DATA_BLOCK "DB3326"
TITLE ==CH2++ZNE05_Alarm_List
{ S7_language := '16(1) Italiano (Italia)  10.08.2015  13:02:09' }
VERSION : 0.1


  STRUCT
   CM_ID : STRING  [8 ] := '=CH2_4';	//IDENTIFICATIVO TRATTO
   STATION_ID : STRING  [8 ] := '++ZNE05';	//TRATTO - ZONA - STAZIONE
   ELEMENT_ID : STRING  [8 ];	//ELEMENTO
   DB_ID : INT  := 3;	//GRANDEZZA DB O TIPO
   PART_IDENTIFICATION : STRING  [12 ];	//IDENTIFICAZIONE PEZZO IN LAVORAZIONE
   ACT_CYCLE_TIME : INT ;	//TEMPO CICLO EFFETTIVO
   COUNT_GOOD : INT ;	//PEZZO PRODOTTO BUONO
   COUNT_SCRAP : INT ;	//PEZZO PRODOTTO DI SCARTO
   ACCUMULATORS : ARRAY  [0 .. 15 ] OF //ACCUMULI
   INT ;
   SPARE_01 : ARRAY  [0 .. 17 ] OF //RISERVE
   INT ;
   CODE_EVENT : ARRAY  [0 .. 7 ] OF //CODICI DI DIAGNOSTICA (codici a 4 cifre)
   INT ;
   EVENTS : STRUCT 	//EVENTI DI DIAGNOSTICA / MONITORAGGIO (bit)
    E0001 : BOOL ;	//=CH2_4++ZNE05+HCZ01-DMC01;FALHA NO MÓDULO ET200S;1
    E0002 : BOOL ;	//=CH2_4++ZNE05+HCZ01-DSW01;FALHA DE SCALANCE;1
    E0003 : BOOL ;	//=CH2_4++ZNE05+HCZ01-QF_06;ALIMENTAÇÃO DISJUNTOR TÉRMICO PARA CIRCUITOS AUXILIARES;1
    E0004 : BOOL ;	//=CH2_4++ZNE05+HCZ01-QF_07;DISJUNTOR TÉRMICO. PODER COMANDOS E SINAIS DE SAÍDA;1
    E0005 : BOOL ;	//=CH2_4++ZNE05+HCZ01-QF_08;FONTE DE ALIMENTAÇÃO MAGNETOTÉRMICA PARA CIRCUITOS DE SEGURANÇA;1
    E0006 : BOOL ;	//=CH2_4++ZNE05+HCZ01-QF_09;DISJUNTOR TÉRMICO. PODER MÓDULOS E SWITCHES E/S ET200;1
    E0007 : BOOL ;
    E0008 : BOOL ;
    E0009 : BOOL ;
    E0010 : BOOL ;
    E0011 : BOOL ;
    E0012 : BOOL ;
    E0013 : BOOL ;
    E0014 : BOOL ;
    E0015 : BOOL ;
    E0016 : BOOL ;
    E0017 : BOOL ;	//=CH2_4++ZNE05+HCZ01-QF_10;FONTE DE ALIMENTAÇÃO 24VDC MOVIFIT FC01-FC02-FC03-FC04;1
    E0018 : BOOL ;	//=CH2_4++ZNE05+HCZ01-QF_11;24Vdc MOVIFIT FC05-06-07-08-09-10 SEP_04;1
    E0019 : BOOL ;	//=CH2_4++ZNE05+HCZ01-QF_20;440Vac MOVIFIT FC01 SETOR MOTOR 1 ZONA 5;1
    E0020 : BOOL ;	//=CH2_4++ZNE05+HCZ01-QF_21;440Vac MOVIFIT FC02 MOTOR SETOR 1 ZONA 5;1
    E0021 : BOOL ;	//=CH2_4++ZNE05+HCZ01-QF_22;FONTE DE ALIMENTAÇÃO 440Vac PARA MOTOR DA PLATAFORMA ESB01 SETOR 1;1
    E0022 : BOOL ;	//=CH2_4++ZNE05+HCZ01-QF_23;440Vac MOVIFIT FC03 MOTOR SETOR 2 ZONA 5;1
    E0023 : BOOL ;	//=CH2_4++ZNE05+HCZ01-QF_24;440Vac MOVIFIT FC04 MOTOR SETOR 3 ZONA 5;1
    E0024 : BOOL ;	//=CH2_4++ZNE05+HCZ01-QF_25;440Vca MOT. MOVIFIT FC05 - 06 - 07 SET. 4 ZONA 5;1
    E0025 : BOOL ;	//=CH2_4++ZNE05+HCZ01-QF_26;FONTE DE ALIMENTAÇÃO 440Vac PARA MOTOR PLATAFORMA ESB02, SETOR 4;1
    E0026 : BOOL ;	//=CH2_4++ZNE05+HCZ01-QF_27;440Vca MOT. MOVIFIT FC08 - 09 - 10 SEMANAS 5 ZONA 5;1
    E0027 : BOOL ;	//=CH2_4++ZNE05+HCZ01-KMS02;MOVIFIT FC01 SETOR DE EFICIÊNCIA DO RELÉ 1;1
    E0028 : BOOL ;	//=CH2_4++ZNE05+HCZ01-KMS04;EFICIÊNCIA DO RELÉ FC02 +ESB01 SETOR 1;1
    E0029 : BOOL ;	//=CH2_4++ZNE05+HCZ01-KMS06;MOVIFIT FC03 SETOR DE EFICIÊNCIA DO RELÉ 2;1
    E0030 : BOOL ;	//=CH2_4++ZNE05+HCZ01-KMS08;MOVIFIT FC04 SETOR DE EFICIÊNCIA DO RELÉ 3;1
    E0031 : BOOL ;	//=CH2_4++ZNE05+HCZ01-KMS010;EFICIÊNCIA DO RELÉ FC05 - 06 - 07 SETOR 4;1
    E0032 : BOOL ;	//=CH2_4++ZNE05+HCZ01-KMS012;EFICIÊNCIA DO RELÉ FC08 - 09 - 10 SETOR 5;1
    E0033 : BOOL ;	//=CH2_4++ZNE05+PTZ01-DMC01;FALHA NO MÓDULO ET200S;1
    E0034 : BOOL ;	//=CH2_4++ZNE05+PTZ02-DMC01;FALHA NO MÓDULO ET200S;1
    E0035 : BOOL ;	//=CH2_4++ZNE05+HKL01-DMC01;FALHA NO MÓDULO ET200S;1
    E0036 : BOOL ;	//=CH2_4++ZNE05+HKL02-DMC01;FALHA NO MÓDULO ET200S;1
    E0037 : BOOL ;	//=CH2_4++ZNE05+PLS01;FALHA DO SCANNER LASER;1
    E0038 : BOOL ;	//=CH2_4++ZNE05+PLS02;FALHA DO SCANNER LASER;1
    E0039 : BOOL ;	//=CH2_4++ZNE05+PLS03;FALHA DO SCANNER LASER;1
    E0040 : BOOL ;	//=CH2_4++ZNE05+PLS04;FALHA DO SCANNER LASER;1
    E0041 : BOOL ;	//=CH2_4++ZNE05+HCZ01-QF_28;FONTE DE ALIMENTAÇÃO 440Vac PARA MOTOR DA PLATAFORMA ESB03 SETOR 1;1
    E0042 : BOOL ;	//=CH2_4++ZNE05+HCZ01-KMS014;ESB03 SETOR DE EFICIÊNCIA DE RELÉ 1;1
    E0043 : BOOL ;	//=CH2_4++ZNE05+XGA01-SC_01;PORTÃO EM ANOMALIA;1
    E0044 : BOOL ;
    E0045 : BOOL ;
    E0046 : BOOL ;
    E0047 : BOOL ;
    E0048 : BOOL ;
    E0049 : BOOL ;
    E0050 : BOOL ;
    E0051 : BOOL ;
    E0052 : BOOL ;
    E0053 : BOOL ;
    E0054 : BOOL ;
    E0055 : BOOL ;
    E0056 : BOOL ;
    E0057 : BOOL ;
    E0058 : BOOL ;
    E0059 : BOOL ;
    E0060 : BOOL ;
    E0061 : BOOL ;
    E0062 : BOOL ;
    E0063 : BOOL ;
    E0064 : BOOL ;
    E0065 : BOOL ;
    E0066 : BOOL ;
    E0067 : BOOL ;
    E0068 : BOOL ;
    E0069 : BOOL ;
    E0070 : BOOL ;
    E0071 : BOOL ;
    E0072 : BOOL ;
    E0073 : BOOL ;
    E0074 : BOOL ;
    E0075 : BOOL ;
    E0076 : BOOL ;
    E0077 : BOOL ;
    E0078 : BOOL ;
    E0079 : BOOL ;
    E0080 : BOOL ;
    E0081 : BOOL ;	//=CH2_4++ZNE05+PTZ01-SB_07;BOTÃO DE EMERGENCIA APERTADO;2
    E0082 : BOOL ;	//=CH2_4++ZNE05+PTZ01-SB_07;EMERGÊNCIA NÃO RESTAURADA;2
    E0083 : BOOL ;	//=CH2_4++ZNE05+PTZ02-SB_07;BOTÃO DE EMERGENCIA APERTADO;2
    E0084 : BOOL ;	//=CH2_4++ZNE05+PTZ02-SB_07;EMERGÊNCIA NÃO RESTAURADA;2
    E0085 : BOOL ;	//=CH2_4++ZNE05+XGA01-SC_01;ACESSO ABERTO NÃO PROGRAMADO (GM);2
    E0086 : BOOL ;	//=CH2_4++ZNE05+XGA01-SC_01;ACESSO NÃO RESTAURADO(GM);2
    E0087 : BOOL ;	//=CH2_4++ZNE05+PRB03-BR_01;BARREIRA INTERDITADA;2
    E0088 : BOOL ;	//=CH2_4++ZNE05+PRB03-BR_01;BARREIRA NÃO RESTAURADA;2
    E0089 : BOOL ;	//=CH2_4++ZNE05+PRB04-BR_02;BARREIRA INTERDITADA;2
    E0090 : BOOL ;	//=CH2_4++ZNE05+PRB04-BR_02;BARREIRA NÃO RESTAURADA;2
    E0091 : BOOL ;	//=CH2_4++ZNE05+PRB01-BR_03;BARREIRA INTERDITADA;2
    E0092 : BOOL ;	//=CH2_4++ZNE05+PRB01-BR_03;BARREIRA NÃO RESTAURADA;2
    E0093 : BOOL ;	//=CH2_4++ZNE05+PRB02-VT_02;BARREIRA INTERDITADA;2
    E0094 : BOOL ;	//=CH2_4++ZNE05+PRB02-VT_02;BARREIRA NÃO RESTAURADA;2
    E0095 : BOOL ;	//=CH2_4++ZNE05+PLS01;SCANNER LASER OCUPADO;2
    E0096 : BOOL ;	//=CH2_4++ZNE05+PLS01;SCANNER LASER NÃO RESTAURADO;2
    E0097 : BOOL ;	//=CH2_4++ZNE05+PLS02;SCANNER LASER OCUPADO;2
    E0098 : BOOL ;	//=CH2_4++ZNE05+PLS02;SCANNER LASER NÃO RESTAURADO;2
    E0099 : BOOL ;	//=CH2_4++ZNE05+PLS03;SCANNER LASER OCUPADO;2
    E0100 : BOOL ;	//=CH2_4++ZNE05+PLS03;SCANNER LASER NÃO RESTAURADO;2
    E0101 : BOOL ;	//=CH2_4++ZNE05+PLS04;SCANNER LASER OCUPADO;2
    E0102 : BOOL ;	//=CH2_4++ZNE05+PLS04;SCANNER LASER NÃO RESTAURADO;2
    E0103 : BOOL ;	//=CH2_4++ZNE05+SLL01-SB_01;BOTÃO DE EMERGENCIA APERTADO;2
    E0104 : BOOL ;	//=CH2_4++ZNE05+SLL01-SB_01;EMERGÊNCIA NÃO RESTAURADA;2
    E0105 : BOOL ;	//=CH2_4++ZNE05+SLL02-SB_01;BOTÃO DE EMERGENCIA APERTADO;2
    E0106 : BOOL ;	//=CH2_4++ZNE05+SLL02-SB_01;EMERGÊNCIA NÃO RESTAURADA;2
    E0107 : BOOL ;	//=CH2_4++ZNE05+PEM01-SB_01;BOTÃO DE EMERGENCIA APERTADO;2
    E0108 : BOOL ;	//=CH2_4++ZNE05+PEM01-SB_01;EMERGÊNCIA NÃO RESTAURADA;2
    E0109 : BOOL ;	//=CH2_4++ZNE05+PEM02-SB_01;BOTÃO DE EMERGENCIA APERTADO;2
    E0110 : BOOL ;	//=CH2_4++ZNE05+PEM02-SB_01;EMERGÊNCIA NÃO RESTAURADA;2
    E0111 : BOOL ;	//=CH2_4++ZNE05+PSC01-SB_01;BOTÃO DE EMERGENCIA APERTADO;2
    E0112 : BOOL ;	//=CH2_4++ZNE05+PSC01-SB_01;EMERGÊNCIA NÃO RESTAURADA;2
    E0113 : BOOL ;	//=CH2_4++ZNE05+PSC02-SB_01;BOTÃO DE EMERGENCIA APERTADO;2
    E0114 : BOOL ;	//=CH2_4++ZNE05+PSC02-SB_01;EMERGÊNCIA NÃO RESTAURADA;2
    E0115 : BOOL ;	//=CH2_4++ZNE05+PSC03-SB_01;BOTÃO DE EMERGENCIA APERTADO;2
    E0116 : BOOL ;	//=CH2_4++ZNE05+PSC03-SB_01;EMERGÊNCIA NÃO RESTAURADA;2
    E0117 : BOOL ;
    E0118 : BOOL ;
    E0119 : BOOL ;	//=CH2_4++ZNE05+XGA01-SC_01;MANUTENÇÃO PROGRAMADA DE ACESSO ABERTO (PM);13
    E0120 : BOOL ;	//=CH2_4++ZNE05+XGA01-SC_01;LIMPEZA TÉCNICA DE ACESSO ABERTO (AM);14
    E0121 : BOOL ;	//=CH2_4++ZNE05+XGA01-SC_01;ACESSO NÃO RESTAURADO PROG. DE MANUTENÇÃO (PM);13
    E0122 : BOOL ;	//=CH2_4++ZNE05+XGA01-SC_01;ACESSO NÃO RESTAURADO LIMPEZA TÉCNICA (AM);14
    E0123 : BOOL ;	//=CH2_4++ZNE05+OIB01-SB_01;BOTÃO DE EMERGENCIA APERTADO;2
    E0124 : BOOL ;	//=CH2_4++ZNE05+OIB01-SB_01;EMERGÊNCIA NÃO RESTAURADA;2
    E0125 : BOOL ;
    E0126 : BOOL ;
    E0127 : BOOL ;
    E0128 : BOOL ;
    E0129 : BOOL ;	//=CH2_4++ZNE05+HCZ01-QF_03;FONTE DE ALIMENTAÇÃO MAGNETOTÉRMICA PARA AR CONDICIONADO 400V;58
    E0130 : BOOL ;	//=CH2_4++ZNE05+HCZ01-QF_15;MAGNETO. PODER PAINEL OPERADOR 24Vdc +PTZ01;58
    E0131 : BOOL ;	//=CH2_4++ZNE05+HCZ01-QF_16;MAGNETO. PODER PAINEL OPERADOR 24Vdc +PTZ02;58
    E0132 : BOOL ;	//=CH2_4++ZNE05+PTZ01-DSP01;PRÉ-ALARME SEM PLC <-> COMUNICAÇÃO IHM;58
    E0133 : BOOL ;	//=CH2_4++ZNE05+PTZ02-DSP01;PRÉ-ALARME SEM PLC <-> COMUNICAÇÃO IHM;58
    E0134 : BOOL ;	//=CH2_4++ZNE05+PTZ01-SA_03;PEDIDO DE ACESSO PARA MANUTENÇÃO PLANEJADA (PM);58
    E0135 : BOOL ;	//=CH2_4++ZNE05+PTZ01-SA_03;SOLICITAR ACESSO PARA LIMPEZA TÉCNICA (AM);58
    E0136 : BOOL ;	//=CH2_4++ZNE05+PTZ02-SA_03;PEDIDO DE ACESSO PARA MANUTENÇÃO PLANEJADA (PM);58
    E0137 : BOOL ;	//=CH2_4++ZNE05+PTZ02-SA_03;SOLICITAR ACESSO PARA LIMPEZA TÉCNICA (AM);58
    E0138 : BOOL ;	//=CH2_4++ZNE05+PTZ01-SA_03;SOLICITAR ACESSO PARA MANUTENÇÃO NÃO PROGRAMADA (GM);58
    E0139 : BOOL ;	//=CH2_4++ZNE05+PTZ02-SA_03;SOLICITAR ACESSO PARA MANUTENÇÃO NÃO PROGRAMADA (GM);58
    E0140 : BOOL ;	//=CH2_4++ZNE05+HCZ01-ST_01;CONTROLE DE TEMPERATURA DO GABINETE;58
    E0141 : BOOL ;	//=CH2_4++ZNE05+PLS01;SCANNER LASER EM PRÉ-ALARME;58
    E0142 : BOOL ;	//=CH2_4++ZNE05+PLS02;SCANNER LASER EM PRÉ-ALARME;58
    E0143 : BOOL ;	//=CH2_4++ZNE05+PLS03;SCANNER LASER EM PRÉ-ALARME;58
    E0144 : BOOL ;	//=CH2_4++ZNE05+PLS04;SCANNER LASER EM PRÉ-ALARME;58
    E0145 : BOOL ;	//=CH2_4++ZNE05+PTZ01;SETOR ASCENTE NÃO ESTÁ EM CICLO INICIADO;58
    E0146 : BOOL ;	//=CH2_4++ZNE05+PTZ01;SETOR JUSANTE NÃO ESTÁ EM CICLO INICIADO;58
    E0147 : BOOL ;	//=CH2_4++ZNE05+PTZ02;SETOR ASCENTE NÃO ESTÁ EM CICLO INICIADO;58
    E0148 : BOOL ;	//=CH2_4++ZNE05+PTZ02;SETOR JUSANTE NÃO ESTÁ EM CICLO INICIADO;58
    E0149 : BOOL ;	//=CH2_4++ZNE05+PTZ03;SETOR ASCENTE NÃO ESTÁ EM CICLO INICIADO;58
    E0150 : BOOL ;	//=CH2_4++ZNE05+PTZ03;SETOR JUSANTE NÃO ESTÁ EM CICLO INICIADO;58
    E0151 : BOOL ;	//=CH2_4++ZNE05+PRE01;SETOR ASCENTE NÃO ESTÁ EM CICLO INICIADO;58
    E0152 : BOOL ;	//=CH2_4++ZNE05+PRE01;SETOR JUSANTE NÃO ESTÁ EM CICLO INICIADO;58
    E0153 : BOOL ;	//=CH2_4++ZNE05+HCZ01;PRÉ-ALARME DE SEGURANÇA DE BYPASS ATIVO;54
    E0154 : BOOL ;	//=CH2_4++ZNE05+TTS06;NKE WARNING TROCA CARTA DE LIMPEZA;4
    E0155 : BOOL ;	//=CH2_4++ZNE05+TTS06;ALARME TROCA DO CARTÃO NKE LIMPEZA;3
    E0156 : BOOL ;	//=CH2_4++ZNE05+LM07;PARCEIRO DE BATERIA DO FIM DE CURSO ACIONADO;10
    E0157 : BOOL ;
    E0158 : BOOL ;
    E0159 : BOOL ;
    E0160 : BOOL ;
    E0161 : BOOL ;
    E0162 : BOOL ;
    E0163 : BOOL ;
    E0164 : BOOL ;
    E0165 : BOOL ;
    E0166 : BOOL ;
    E0167 : BOOL ;
    E0168 : BOOL ;
    E0169 : BOOL ;
    E0170 : BOOL ;
    E0171 : BOOL ;
    E0172 : BOOL ;
    E0173 : BOOL ;
    E0174 : BOOL ;
    E0175 : BOOL ;
    E0176 : BOOL ;
    E0177 : BOOL ;	//=CH2_4++ZNE05+OIB01-DMC01;ANOMALIA DO MÓDULO ProfSafe ET200S-FDI-FDO;2
    E0178 : BOOL ;	//=CH2_4++ZNE05+HCZ01-DMC01;ANOMALIA DO MÓDULO ProfSafe ET200S-FDI-FDO;2
    E0179 : BOOL ;	//=CH2_4++ZNE05+PTZ01-DMC01;ANOMALIA DO MÓDULO ProfSafe ET200S-FDI;2
    E0180 : BOOL ;	//=CH2_4++ZNE05+PTZ02-DMC01;ANOMALIA DO MÓDULO ProfSafe ET200S-FDI;2
    E0181 : BOOL ;	//=CH2_4++ZNE05+PTZ03-DMC01;ANOMALIA DO MÓDULO ProfSafe ET200S-FDI;2
    E0182 : BOOL ;	//=CH2_4++ZNE05+PRE01-DMC01;ANOMALIA DO MÓDULO ProfSafe ET200S-FDI;2
    E0183 : BOOL ;	//=CH2_4++ZNE05+HKL01-DMC01;ANOMALIA DO MÓDULO ProfSafe ET200S-FDI;2
    E0184 : BOOL ;	//=CH2_4++ZNE05+HKL02-DMC01;ANOMALIA DO MÓDULO ProfSafe ET200S-FDI;2
    E0185 : BOOL ;	//=CH2_4++ZNE05+HCZ02-DMC01;ANOMALIA DO MÓDULO ProfSafe ET200S-FDI-FDO;2
    E0186 : BOOL ;
    E0187 : BOOL ;
    E0188 : BOOL ;
    E0189 : BOOL ;
    E0190 : BOOL ;
    E0191 : BOOL ;
    E0192 : BOOL ;
    E0193 : BOOL ;
    E0194 : BOOL ;
    E0195 : BOOL ;
    E0196 : BOOL ;
    E0197 : BOOL ;
    E0198 : BOOL ;
    E0199 : BOOL ;
    E0200 : BOOL ;
    E0201 : BOOL ;
    E0202 : BOOL ;
    E0203 : BOOL ;
    E0204 : BOOL ;
    E0205 : BOOL ;
    E0206 : BOOL ;
    E0207 : BOOL ;
    E0208 : BOOL ;
    E0209 : BOOL ;	//=CH2_4++ZNE05;EM PRODUÇÃO;19
    E0210 : BOOL ;	//=CH2_4++ZNE05+PTZ01-SB_05;INICIAR CICLO AUTOMÁTICO;15
    E0211 : BOOL ;	//=CH2_4++ZNE05+PTZ02-SB_05;INICIAR CICLO AUTOMÁTICO;15
    E0212 : BOOL ;	//=CH2_4++ZNE05+PTZ01-SA_01;CICLO MANUAL SELECIONADO;16
    E0213 : BOOL ;	//=CH2_4++ZNE05+PTZ02-SA_01;CICLO MANUAL SELECIONADO;16
    E0214 : BOOL ;	//=CH2_4++ZNE05+PTZ01-SB_04;PARADA DO CICLO;17
    E0215 : BOOL ;	//=CH2_4++ZNE05+PTZ02-SB_04;PARADA DO CICLO;17
    E0216 : BOOL ;
    E0217 : BOOL ;	//=CH2_4++ZNE05+TTS01;FALHA NO CARREGAMENTO;6
    E0218 : BOOL ;	//=CH2_4++ZNE05+TTS12;FALHA NO DESCARREGAMENTO;9
    E0219 : BOOL ;	//=CH2_4++ZNE05+TTS04;OPERADOR DE SOBRECICLO;8
    E0220 : BOOL ;	//=CH2_4++ZNE05+TTS05;OPERADOR DE SOBRECICLO;8
    E0221 : BOOL ;
    E0222 : BOOL ;
    E0223 : BOOL ;
    E0224 : BOOL ;
    E0225 : BOOL ;	//=CH2_4++ZNE05+TTS01-SQA01;FALHA NO INTERRUPTOR DE LIMITE DE PARADA;1
    E0226 : BOOL ;	//=CH2_4++ZNE05+TTS01-SQS01;FALHA NO INTERRUPTOR DE LIMITE DE LENTAÇÃO;1
    E0227 : BOOL ;	//=CH2_4++ZNE05+TTS01-SQC01;FALHA NO INTERRUPTOR DE LIMITE DE CONTROLE DE POSIÇÃO;1
    E0228 : BOOL ;	//=CH2_4++ZNE05+TTS01-B__01;FALHA DA FOTOCÉLULA NA PRESENÇA DO VEÍCULO;1
    E0229 : BOOL ;	//=CH2_4++ZNE05+TTS01;SAIR DO TEMPO DE TRANSFERÊNCIA;1
    E0230 : BOOL ;	//=CH2_4++ZNE05+TTS01;CTRL ENGRENAGEM TTS ANTERIOR;1
    E0231 : BOOL ;	//=CH2_4++ZNE05+TTS01;CTRL ENGRENAGEM PRÓXIMO TTS;1
    E0232 : BOOL ;	//=CH2_4++ZNE05+TTS01;POSIÇÃO CTRL;1
    E0233 : BOOL ;	//=CH2_4++ZNE05+TTS01-M__01;FALHA NO INVERSOR;1
    E0234 : BOOL ;	//=CH2_4++ZNE05+TTS01-M__01;ERRO DE COMUNICAÇÃO DO INVERSOR;1
    E0235 : BOOL ;	//=CH2_4++ZNE05+TTS01-SQA02;FALHA DO INTERRUPTOR DE LIMITE DE PROTEÇÃO QUEDA TRABALHO FECHADO;1
    E0236 : BOOL ;	//=CH2_4++ZNE05+TTS01-SQB02;FALHA DE RESTO ABERTO DO INTERRUPTOR DE LIMITE DE PROTEÇÃO QUEDA;1
    E0237 : BOOL ;	//=CH2_4++ZNE05+TTS01-SQ_01;QUEBRA DA CORREIA DE TRANSMISSÃO TTS;1
    E0238 : BOOL ;	//=CH2_4++ZNE05+TTS01;PRÉ-ALARME DE BYPASS DE FALHA ATIVO;58
    E0239 : BOOL ;	//=CH2_4++ZNE05+TTS01-M__01;PRÉ-ALARME DE CORRENTE ABSORVIDA;58
    E0240 : BOOL ;	//=CH2_4++ZNE05+TTS01-M__01;PRÉ-ALARME DO INVERSOR MOVIMOT;58
    E0241 : BOOL ;	//=CH2_4++ZNE05+TTS01-U__01;ERRO DE COMUNICAÇÃO MOVIFIT;1
    E0242 : BOOL ;	//=CH2_4++ZNE05+TTS01-U__01;INTERRUPTOR MOVIFIT ABERTO 380V;1
    E0243 : BOOL ;	//=CH2_4++ZNE05+TTS01-U__01;AUSÊNCIAS 24 VOLTS MOVIFIT SEGURANÇA;1
    E0244 : BOOL ;	//=CH2_4++ZNE05+TTS01-U__01;AUSÊNCIAS MOVIFIT 24 VOLT;1
    E0245 : BOOL ;	//=CH2_4++ZNE05+TTS01-U__01;ANOMALIA MOVIFIT;1
    E0246 : BOOL ;	//=CH2_4++ZNE05+TTS01-U__01;SOBRECARGA DE TENSÃO DE SAÍDA 0 MOVIFIT;1
    E0247 : BOOL ;	//=CH2_4++ZNE05+TTS01-U__01;TENSÃO DE SAÍDA DE SOBRECARGA SAÍDA 1 MOVIFIT;1
    E0248 : BOOL ;	//=CH2_4++ZNE05+TTS01-U__01;SOBRECARGA DE TENSÃO DO MOVIFIT NA SAÍDA 2;1
    E0249 : BOOL ;	//=CH2_4++ZNE05+TTS01-U__01;SOBRECARGA DE TENSÃO DE SAÍDA 3 MOVIFIT;1
    E0250 : BOOL ;	//=CH2_4++ZNE05+TTS01-U__01;SOBRECARGA DE TENSÃO DO SENSOR MOVIFIT GRUPO 1;1
    E0251 : BOOL ;	//=CH2_4++ZNE05+TTS01-U__01;SOBRECARGA DE TENSÃO DO SENSOR MOVIFIT GRUPO 2;1
    E0252 : BOOL ;	//=CH2_4++ZNE05+TTS01-U__01;SOBRECARGA DE TENSÃO DO SENSOR MOVIFIT GRUPO 3;1
    E0253 : BOOL ;	//=CH2_4++ZNE05+TTS01-U__01;SOBRECARGA DE TENSÃO DO SENSOR MOVIFIT GRUPO 4;1
    E0254 : BOOL ;
    E0255 : BOOL ;
    E0256 : BOOL ;
    E0257 : BOOL ;	//=CH2_4++ZNE05+TTS02-SQA01;FALHA NO INTERRUPTOR DE LIMITE DE PARADA;1
    E0258 : BOOL ;	//=CH2_4++ZNE05+TTS02-SQS01;FALHA NO INTERRUPTOR DE LIMITE DE LENTAÇÃO;1
    E0259 : BOOL ;	//=CH2_4++ZNE05+TTS02-SQC01;FALHA NO INTERRUPTOR DE LIMITE DE CONTROLE DE POSIÇÃO;1
    E0260 : BOOL ;	//=CH2_4++ZNE05+TTS02-B__01;FALHA DA FOTOCÉLULA NA PRESENÇA DO VEÍCULO;1
    E0261 : BOOL ;	//=CH2_4++ZNE05+TTS02;SAIR DO TEMPO DE TRANSFERÊNCIA;1
    E0262 : BOOL ;	//=CH2_4++ZNE05+TTS02;CTRL ENGRENAGEM TTS ANTERIOR;1
    E0263 : BOOL ;	//=CH2_4++ZNE05+TTS02;CTRL ENGRENAGEM PRÓXIMO TTS;1
    E0264 : BOOL ;	//=CH2_4++ZNE05+TTS02;POSIÇÃO CTRL;1
    E0265 : BOOL ;	//=CH2_4++ZNE05+TTS02-M__01;FALHA NO INVERSOR;1
    E0266 : BOOL ;	//=CH2_4++ZNE05+TTS02-M__01;ERRO DE COMUNICAÇÃO DO INVERSOR;1
    E0267 : BOOL ;	//=CH2_4++ZNE05+TTS02-SQA02;FALHA DO INTERRUPTOR DE LIMITE DE PROTEÇÃO QUEDA TRABALHO FECHADO;1
    E0268 : BOOL ;	//=CH2_4++ZNE05+TTS02-SQB02;FALHA DE RESTO ABERTO DO INTERRUPTOR DE LIMITE DE PROTEÇÃO QUEDA;1
    E0269 : BOOL ;	//=CH2_4++ZNE05+TTS02-SQ_01;QUEBRA DA CORREIA DE TRANSMISSÃO TTS;1
    E0270 : BOOL ;	//=CH2_4++ZNE05+TTS02;PRÉ-ALARME DE BYPASS DE FALHA ATIVO;58
    E0271 : BOOL ;	//=CH2_4++ZNE05+TTS02-M__01;PRÉ-ALARME DE CORRENTE ABSORVIDA;58
    E0272 : BOOL ;	//=CH2_4++ZNE05+TTS02-M__01;PRÉ-ALARME DO INVERSOR MOVIMOT;58
    E0273 : BOOL ;	//=CH2_4++ZNE05+TTS02-U__01;ERRO DE COMUNICAÇÃO MOVIFIT;1
    E0274 : BOOL ;	//=CH2_4++ZNE05+TTS02-U__01;INTERRUPTOR MOVIFIT ABERTO 380V;1
    E0275 : BOOL ;	//=CH2_4++ZNE05+TTS02-U__01;AUSÊNCIAS 24 VOLTS MOVIFIT SEGURANÇA;1
    E0276 : BOOL ;	//=CH2_4++ZNE05+TTS02-U__01;AUSÊNCIAS MOVIFIT 24 VOLT;1
    E0277 : BOOL ;	//=CH2_4++ZNE05+TTS02-U__01;ANOMALIA MOVIFIT;1
    E0278 : BOOL ;	//=CH2_4++ZNE05+TTS02-U__01;SOBRECARGA DE TENSÃO DE SAÍDA 0 MOVIFIT;1
    E0279 : BOOL ;	//=CH2_4++ZNE05+TTS02-U__01;TENSÃO DE SAÍDA DE SOBRECARGA SAÍDA 1 MOVIFIT;1
    E0280 : BOOL ;	//=CH2_4++ZNE05+TTS02-U__01;SOBRECARGA DE TENSÃO DO MOVIFIT NA SAÍDA 2;1
    E0281 : BOOL ;	//=CH2_4++ZNE05+TTS02-U__01;SOBRECARGA DE TENSÃO DE SAÍDA 3 MOVIFIT;1
    E0282 : BOOL ;	//=CH2_4++ZNE05+TTS02-U__01;SOBRECARGA DE TENSÃO DO SENSOR MOVIFIT GRUPO 1;1
    E0283 : BOOL ;	//=CH2_4++ZNE05+TTS02-U__01;SOBRECARGA DE TENSÃO DO SENSOR MOVIFIT GRUPO 2;1
    E0284 : BOOL ;	//=CH2_4++ZNE05+TTS02-U__01;SOBRECARGA DE TENSÃO DO SENSOR MOVIFIT GRUPO 3;1
    E0285 : BOOL ;	//=CH2_4++ZNE05+TTS02-U__01;SOBRECARGA DE TENSÃO DO SENSOR MOVIFIT GRUPO 4;1
    E0286 : BOOL ;
    E0287 : BOOL ;
    E0288 : BOOL ;
    E0289 : BOOL ;	//=CH2_4++ZNE05+ESB01-SQA01;FALHA NO INTERRUPTOR DE LIMITE DE PARAGEM INFERIOR DA PLATAFORMA MÓVEL +ESB;1
    E0290 : BOOL ;	//=CH2_4++ZNE05+ESB01-SQB01;FALHA NO INTERRUPTOR DE LIMITE DE PARADA ALTA DA PLATAFORMA MÓVEL +ESB;1
    E0291 : BOOL ;
    E0292 : BOOL ;
    E0293 : BOOL ;	//=CH2_4++ZNE05+ESB01-SQA01;TIME OUT DESCIDA +ESB;1
    E0294 : BOOL ;	//=CH2_4++ZNE05+ESB01-SQB01;TIME OUT RISE +ESB;1
    E0295 : BOOL ;
    E0296 : BOOL ;
    E0297 : BOOL ;	//=CH2_4++ZNE05+ESB01-HKM03;SONDA TÉRMICA DO MOTOR +ESB;1
    E0298 : BOOL ;
    E0299 : BOOL ;
    E0300 : BOOL ;
    E0301 : BOOL ;
    E0302 : BOOL ;
    E0303 : BOOL ;
    E0304 : BOOL ;
    E0305 : BOOL ;	//=CH2_4++ZNE05+ESB01;ESTAÇÃO EXCLUÍDA PRÉ-ALARME;58
    E0306 : BOOL ;
    E0307 : BOOL ;
    E0308 : BOOL ;
    E0309 : BOOL ;
    E0310 : BOOL ;
    E0311 : BOOL ;
    E0312 : BOOL ;
    E0313 : BOOL ;	//=CH2_4++ZNE05+ESB01;PRÉ-ALARME DE BYPASS DE FALHA ATIVO;58
    E0314 : BOOL ;
    E0315 : BOOL ;
    E0316 : BOOL ;
    E0317 : BOOL ;
    E0318 : BOOL ;
    E0319 : BOOL ;
    E0320 : BOOL ;
    E0321 : BOOL ;	//=CH2_4++ZNE05+TTS03-SQA01;FALHA NO INTERRUPTOR DE LIMITE DE PARADA;1
    E0322 : BOOL ;	//=CH2_4++ZNE05+TTS03-SQS01;FALHA NO INTERRUPTOR DE LIMITE DE LENTAÇÃO;1
    E0323 : BOOL ;	//=CH2_4++ZNE05+TTS03-SQC01;FALHA NO INTERRUPTOR DE LIMITE DE CONTROLE DE POSIÇÃO;1
    E0324 : BOOL ;	//=CH2_4++ZNE05+TTS03-B__01;FALHA DA FOTOCÉLULA NA PRESENÇA DO VEÍCULO;1
    E0325 : BOOL ;	//=CH2_4++ZNE05+TTS03;SAIR DO TEMPO DE TRANSFERÊNCIA;1
    E0326 : BOOL ;	//=CH2_4++ZNE05+TTS03;CTRL ENGRENAGEM TTS ANTERIOR;1
    E0327 : BOOL ;	//=CH2_4++ZNE05+TTS03;CTRL ENGRENAGEM PRÓXIMO TTS;1
    E0328 : BOOL ;	//=CH2_4++ZNE05+TTS03;POSIÇÃO CTRL;1
    E0329 : BOOL ;	//=CH2_4++ZNE05+TTS03-M__01;FALHA NO INVERSOR;1
    E0330 : BOOL ;	//=CH2_4++ZNE05+TTS03-M__01;ERRO DE COMUNICAÇÃO DO INVERSOR;1
    E0331 : BOOL ;	//=CH2_4++ZNE05+TTS03-SQA02;FALHA DO INTERRUPTOR DE LIMITE DE PROTEÇÃO QUEDA TRABALHO FECHADO;1
    E0332 : BOOL ;	//=CH2_4++ZNE05+TTS03-SQB02;FALHA DE RESTO ABERTO DO INTERRUPTOR DE LIMITE DE PROTEÇÃO QUEDA;1
    E0333 : BOOL ;	//=CH2_4++ZNE05+TTS03-SQ_01;QUEBRA DA CORREIA DE TRANSMISSÃO TTS;1
    E0334 : BOOL ;	//=CH2_4++ZNE05+TTS03;PRÉ-ALARME DE BYPASS DE FALHA ATIVO;58
    E0335 : BOOL ;	//=CH2_4++ZNE05+TTS03-M__01;PRÉ-ALARME DE CORRENTE ABSORVIDA;58
    E0336 : BOOL ;	//=CH2_4++ZNE05+TTS03-M__01;PRÉ-ALARME DO INVERSOR MOVIMOT;58
    E0337 : BOOL ;	//=CH2_4++ZNE05+TTS03-U__01;ERRO DE COMUNICAÇÃO MOVIFIT;1
    E0338 : BOOL ;	//=CH2_4++ZNE05+TTS03-U__01;INTERRUPTOR MOVIFIT ABERTO 380V;1
    E0339 : BOOL ;	//=CH2_4++ZNE05+TTS03-U__01;AUSÊNCIAS 24 VOLTS MOVIFIT SEGURANÇA;1
    E0340 : BOOL ;	//=CH2_4++ZNE05+TTS03-U__01;AUSÊNCIAS MOVIFIT 24 VOLT;1
    E0341 : BOOL ;	//=CH2_4++ZNE05+TTS03-U__01;ANOMALIA MOVIFIT;1
    E0342 : BOOL ;	//=CH2_4++ZNE05+TTS03-U__01;SOBRECARGA DE TENSÃO DE SAÍDA 0 MOVIFIT;1
    E0343 : BOOL ;	//=CH2_4++ZNE05+TTS03-U__01;TENSÃO DE SAÍDA DE SOBRECARGA SAÍDA 1 MOVIFIT;1
    E0344 : BOOL ;	//=CH2_4++ZNE05+TTS03-U__01;SOBRECARGA DE TENSÃO DO MOVIFIT NA SAÍDA 2;1
    E0345 : BOOL ;	//=CH2_4++ZNE05+TTS03-U__01;SOBRECARGA DE TENSÃO DE SAÍDA 3 MOVIFIT;1
    E0346 : BOOL ;	//=CH2_4++ZNE05+TTS03-U__01;SOBRECARGA DE TENSÃO DO SENSOR MOVIFIT GRUPO 1;1
    E0347 : BOOL ;	//=CH2_4++ZNE05+TTS03-U__01;SOBRECARGA DE TENSÃO DO SENSOR MOVIFIT GRUPO 2;1
    E0348 : BOOL ;	//=CH2_4++ZNE05+TTS03-U__01;SOBRECARGA DE TENSÃO DO SENSOR MOVIFIT GRUPO 3;1
    E0349 : BOOL ;	//=CH2_4++ZNE05+TTS03-U__01;SOBRECARGA DE TENSÃO DO SENSOR MOVIFIT GRUPO 4;1
    E0350 : BOOL ;
    E0351 : BOOL ;
    E0352 : BOOL ;
    E0353 : BOOL ;	//=CH2_4++ZNE05+TTS04-SQA01;FALHA NO INTERRUPTOR DE LIMITE DE PARADA;1
    E0354 : BOOL ;	//=CH2_4++ZNE05+TTS04-SQS01;FALHA NO INTERRUPTOR DE LIMITE DE LENTAÇÃO;1
    E0355 : BOOL ;	//=CH2_4++ZNE05+TTS04-SQC01;FALHA NO INTERRUPTOR DE LIMITE DE CONTROLE DE POSIÇÃO;1
    E0356 : BOOL ;	//=CH2_4++ZNE05+TTS04-B__01;FALHA DA FOTOCÉLULA NA PRESENÇA DO VEÍCULO;1
    E0357 : BOOL ;	//=CH2_4++ZNE05+TTS04;SAIR DO TEMPO DE TRANSFERÊNCIA;1
    E0358 : BOOL ;	//=CH2_4++ZNE05+TTS04;CTRL ENGRENAGEM TTS ANTERIOR;1
    E0359 : BOOL ;	//=CH2_4++ZNE05+TTS04;CTRL ENGRENAGEM PRÓXIMO TTS;1
    E0360 : BOOL ;	//=CH2_4++ZNE05+TTS04;POSIÇÃO CTRL;1
    E0361 : BOOL ;	//=CH2_4++ZNE05+TTS04-M__01;FALHA NO INVERSOR;1
    E0362 : BOOL ;	//=CH2_4++ZNE05+TTS04-M__01;ERRO DE COMUNICAÇÃO DO INVERSOR;1
    E0363 : BOOL ;	//=CH2_4++ZNE05+TTS04-SQA02;FALHA DO INTERRUPTOR DE LIMITE DE PROTEÇÃO QUEDA TRABALHO FECHADO;1
    E0364 : BOOL ;	//=CH2_4++ZNE05+TTS04-SQB02;FALHA DE RESTO ABERTO DO INTERRUPTOR DE LIMITE DE PROTEÇÃO QUEDA;1
    E0365 : BOOL ;	//=CH2_4++ZNE05+TTS04-SQ_01;QUEBRA DA CORREIA DE TRANSMISSÃO TTS;1
    E0366 : BOOL ;	//=CH2_4++ZNE05+TTS04;PRÉ-ALARME DE BYPASS DE FALHA ATIVO;58
    E0367 : BOOL ;	//=CH2_4++ZNE05+TTS04-M__01;PRÉ-ALARME DE CORRENTE ABSORVIDA;58
    E0368 : BOOL ;	//=CH2_4++ZNE05+TTS04-M__01;PRÉ-ALARME DO INVERSOR MOVIMOT;58
    E0369 : BOOL ;	//=CH2_4++ZNE05+TTS04-U__01;ERRO DE COMUNICAÇÃO MOVIFIT;1
    E0370 : BOOL ;	//=CH2_4++ZNE05+TTS04-U__01;INTERRUPTOR MOVIFIT ABERTO 380V;1
    E0371 : BOOL ;	//=CH2_4++ZNE05+TTS04-U__01;AUSÊNCIAS 24 VOLTS MOVIFIT SEGURANÇA;1
    E0372 : BOOL ;	//=CH2_4++ZNE05+TTS04-U__01;AUSÊNCIAS MOVIFIT 24 VOLT;1
    E0373 : BOOL ;	//=CH2_4++ZNE05+TTS04-U__01;ANOMALIA MOVIFIT;1
    E0374 : BOOL ;	//=CH2_4++ZNE05+TTS04-U__01;SOBRECARGA DE TENSÃO DE SAÍDA 0 MOVIFIT;1
    E0375 : BOOL ;	//=CH2_4++ZNE05+TTS04-U__01;TENSÃO DE SAÍDA DE SOBRECARGA SAÍDA 1 MOVIFIT;1
    E0376 : BOOL ;	//=CH2_4++ZNE05+TTS04-U__01;SOBRECARGA DE TENSÃO DO MOVIFIT NA SAÍDA 2;1
    E0377 : BOOL ;	//=CH2_4++ZNE05+TTS04-U__01;SOBRECARGA DE TENSÃO DE SAÍDA 3 MOVIFIT;1
    E0378 : BOOL ;	//=CH2_4++ZNE05+TTS04-U__01;SOBRECARGA DE TENSÃO DO SENSOR MOVIFIT GRUPO 1;1
    E0379 : BOOL ;	//=CH2_4++ZNE05+TTS04-U__01;SOBRECARGA DE TENSÃO DO SENSOR MOVIFIT GRUPO 2;1
    E0380 : BOOL ;	//=CH2_4++ZNE05+TTS04-U__01;SOBRECARGA DE TENSÃO DO SENSOR MOVIFIT GRUPO 3;1
    E0381 : BOOL ;	//=CH2_4++ZNE05+TTS04-U__01;SOBRECARGA DE TENSÃO DO SENSOR MOVIFIT GRUPO 4;1
    E0382 : BOOL ;
    E0383 : BOOL ;
    E0384 : BOOL ;
    E0385 : BOOL ;	//=CH2_4++ZNE05+WIP01;PARADA DE LINHA DO MES/PLC PARA CHAMADA DE OPERADOR;11
    E0386 : BOOL ;	//=CH2_4++ZNE05+WIP01;NÓ PROFINET DO LEITOR NÃO ESTÁ OK;1
    E0387 : BOOL ;	//=CH2_4++ZNE05+WIP01;PLACA CODIFICADORA DE NÓ PROFINET NÃO OK;1
    E0388 : BOOL ;	//=CH2_4++ZNE05+WIP01;MAU FUNCIONAMENTO DO SENSOR DE PITCHING;1
    E0389 : BOOL ;	//=CH2_4++ZNE05+WIP01;DISFUNÇÃO DE TRÂNSITO DO PONTO DE AJUSTE;1
    E0390 : BOOL ;	//=CH2_4++ZNE05+WIP01;MAU FUNCIONAMENTO DO CODIFICADOR;1
    E0391 : BOOL ;
    E0392 : BOOL ;
    E0393 : BOOL ;	//=CH2_4++ZNE05+WIP01;ANOMALIA DE LEITURA DE CÓDIGO DE BARRAS/TAG;5
    E0394 : BOOL ;	//=CH2_4++ZNE05+WIP01;TEMPO ESGOTADO DE LEITURA DE CÓDIGO DE BARRAS/TAG;5
    E0395 : BOOL ;	//=CH2_4++ZNE05+WIP01;INCONSISTÊNCIA FÍSICO-LÓGICA;5
    E0396 : BOOL ;	//=CH2_4++ZNE05+WIP01;VERIFIQUE O DÍGITO ERRADO CIS;5
    E0397 : BOOL ;	//=CH2_4++ZNE05+WIP01;TEMPO LIMITE PARA RECEBIMENTO DE DADOS DO PERÍODO ANTERIOR;5
    E0398 : BOOL ;	//=CH2_4++ZNE05+WIP01;INCONSISTÊNCIA DE DADOS DE SET POINT CIS/VIS COM CIS/VIS NEXT;5
    E0399 : BOOL ;	//=CH2_4++ZNE05+WIP01;LINHA WIP DO SERVIÇO MES NÃO ATIVA (PARADA DE LINHA);10
    E0400 : BOOL ;	//=CH2_4++ZNE05+WIP01;NOK PARA CONTINUAR DA ESTAÇÃO AUTOMÁTICA MES (SASERVICE);10
    E0401 : BOOL ;	//=CH2_4++ZNE05+WIP01;SERVIÇO MES SET POINT NÃO ATIVO;58
    E0402 : BOOL ;	//=CH2_4++ZNE05+WIP01;SERVIÇO WIP DRAW MES NÃO ATIVO;58
    E0403 : BOOL ;	//=CH2_4++ZNE05+WIP01;CONFIGURANDO SERVIÇO MES DA ESTAÇÃO NÃO ATIVO;58
    E0404 : BOOL ;	//=CH2_4++ZNE05+WIP01;SERVIÇO DE CHAMADA DE OPERADOR MES;58
    E0405 : BOOL ;	//=CH2_4++ZNE05+WIP01;SERVIÇO DE ESTAÇÃO DE ENVIO DE DADOS MES SASERVICE NÃO ATIVO;58
    E0406 : BOOL ;	//=CH2_4++ZNE05+WIP01;SERVIÇO DA ESTAÇÃO DE SOLICITAÇÃO DE DADOS DO MES SRSERVICE NÃO ATIVO;10
    E0407 : BOOL ;	//=CH2_4++ZNE05+WIP01;MES SMSERVICE ESTAÇÃO MODELO SERVIÇO NÃO ATIVO;58
    E0408 : BOOL ;
    E0409 : BOOL ;	//=CH2_4++ZNE05+WIP01;ESTAÇÃO NÃO EM AUTOMÁTICA;16
    E0410 : BOOL ;	//=CH2_4++ZNE05+WIP01;LEITOR CIS-NEXT BY-PASS DO MES;55
    E0411 : BOOL ;	//=CH2_4++ZNE05+WIP01;ESTAÇÃO EXCLUÍDA;17
    E0412 : BOOL ;	//=CH2_4++ZNE05+WIP01;NEGÓCIO WIP EM MUDANÇA;17
    E0413 : BOOL ;	//=CH2_4++ZNE05+WIP01;RESOLVER CHAMADA DE OPERADOR DO MES/PLC (COGUMELO AMARELO);53
    E0414 : BOOL ;
    E0415 : BOOL ;	//=CH2_4++ZNE05+WIP01;LISTA DE ESTAÇÕES DE CONFIGURAÇÃO VAZIA;10
    E0416 : BOOL ;	//=CH2_4++ZNE05+WIP01;LINHA PARADA POR MÊS;17
    E0417 : BOOL ;	//=CH2_4++ZNE05+LMN01-DSP01;OPERADOR CHAMADA LIMO 01 ESTAÇÃO 82 SX;53
    E0418 : BOOL ;	//=CH2_4++ZNE05+LMN03-DSP01;OPERADOR CHAMADA LIMO 03 ESTAÇÃO 83 SX;53
    E0419 : BOOL ;	//=CH2_4++ZNE05+LMN05-DSP01;OPERADOR CHAMADA LIMO 05 ESTAÇÃO 84 SX;53
    E0420 : BOOL ;	//=CH2_4++ZNE05+LMN07-DSP01;OPERADOR CHAMADA LIMO 07 ESTAÇÃO 85 SX;53
    E0421 : BOOL ;	//=CH2_4++ZNE05+LMN09-DSP01;OPERADOR CHAMADA LIMO 09 ESTAÇÃO 86 SX;53
    E0422 : BOOL ;	//=CH2_4++ZNE05+LMN11-DSP01;OPERADOR CHAMADA LIMO 11 ESTAÇÃO 83A ESQUERDA;53
    E0423 : BOOL ;
    E0424 : BOOL ;
    E0425 : BOOL ;	//=CH2_4++ZNE05+LMN02-DSP01;OPERADOR CHAMADA LIMO 02 ESTAÇÃO 82 DX;53
    E0426 : BOOL ;	//=CH2_4++ZNE05+LMN04-DSP01;OPERADOR CHAMADA LIMO 04 ESTAÇÃO 83 DX;53
    E0427 : BOOL ;	//=CH2_4++ZNE05+LMN06-DSP01;OPERADOR CHAMADA LIMO 06 ESTAÇÃO 84 DX;53
    E0428 : BOOL ;	//=CH2_4++ZNE05+LMN08-DSP01;OPERADOR CHAMADA LIMO 08 ESTAÇÃO 85 DX;53
    E0429 : BOOL ;	//=CH2_4++ZNE05+LMN10-DSP01;CHAMADA DE OPERADOR LIMO 10 ESTAÇÃO 86 DX;53
    E0430 : BOOL ;	//=CH2_4++ZNE05+LMN12-DSP01;OPERADOR CHAMADA LIMO 12 ESTAÇÃO 83A DIREITA;53
    E0431 : BOOL ;
    E0432 : BOOL ;
    E0433 : BOOL ;	//=CH2_4++ZNE05+LMN01-DSP01;PARADA LATERAL DO SILT LINE 01 ESTAÇÃO 82 ESQUERDA;12
    E0434 : BOOL ;	//=CH2_4++ZNE05+LMN03-DSP01;PARADA LADO DA LINHA DE LODO 03 ESTAÇÃO 83 ESQUERDA;12
    E0435 : BOOL ;	//=CH2_4++ZNE05+LMN05-DSP01;PARADA LATERAL DO SILT LINE 05 ESTAÇÃO 84 ESQUERDA;12
    E0436 : BOOL ;	//=CH2_4++ZNE05+LMN07-DSP01;PARADA LATERAL DO SILT LINE 07 ESTAÇÃO 85 ESQUERDA;12
    E0437 : BOOL ;	//=CH2_4++ZNE05+LMN09-DSP01;PARADA LATERAL DO SILT LINE 09 ESTAÇÃO 86 ESQUERDA;12
    E0438 : BOOL ;	//=CH2_4++ZNE05+LMN11-DSP01;PARADA LADO DA LINHA DE SILT 11 ESTAÇÃO 83A ESQUERDA;12
    E0439 : BOOL ;
    E0440 : BOOL ;
    E0441 : BOOL ;	//=CH2_4++ZNE05+LMN02-DSP01;PARADA LADO DA LINHA DE LODO 02 ESTAÇÃO 82 DIREITA;12
    E0442 : BOOL ;	//=CH2_4++ZNE05+LMN04-DSP01;PARADA LADO DA LINHA DE LODO 04 ESTAÇÃO 83 DIREITA;12
    E0443 : BOOL ;	//=CH2_4++ZNE05+LMN06-DSP01;PARADA LADO DA LINHA DE LODO 06 ESTAÇÃO 84 DIREITA;12
    E0444 : BOOL ;	//=CH2_4++ZNE05+LMN08-DSP01;PARADA LADO DA LINHA DE SILT 08 ESTAÇÃO 85 DIREITA;12
    E0445 : BOOL ;	//=CH2_4++ZNE05+LMN10-DSP01;PARADA LADO DA LINHA DE SILT 10 ESTAÇÃO 86 DIREITA;12
    E0446 : BOOL ;	//=CH2_4++ZNE05+LMN12-DSP01;PARADA LADO DA LINHA DE SILT 12 ESTAÇÃO 83A DIREITA;12
    E0447 : BOOL ;
    E0448 : BOOL ;
    E0449 : BOOL ;	//=CH2_4++ZNE05+HCZ02-DMC01;FALHA NO MÓDULO ET200S;1
    E0450 : BOOL ;	//=CH2_4++ZNE05+HCZ02-DSW01;FALHA DE SCALANCE;1
    E0451 : BOOL ;	//=CH2_4++ZNE05+HCZ02-QF_06;ALIMENTAÇÃO DISJUNTOR TÉRMICO PARA CIRCUITOS AUXILIARES;1
    E0452 : BOOL ;	//=CH2_4++ZNE05+HCZ02-QF_07;DISJUNTOR TÉRMICO. PODER COMANDOS E SINAIS DE SAÍDA;1
    E0453 : BOOL ;	//=CH2_4++ZNE05+HCZ02-QF_08;FONTE DE ALIMENTAÇÃO MAGNETOTÉRMICA PARA CIRCUITOS DE SEGURANÇA;1
    E0454 : BOOL ;	//=CH2_4++ZNE05+HCZ02-QF_09;DISJUNTOR TÉRMICO. PODER MÓDULOS E SWITCHES E/S ET200;1
    E0455 : BOOL ;
    E0456 : BOOL ;
    E0457 : BOOL ;
    E0458 : BOOL ;
    E0459 : BOOL ;
    E0460 : BOOL ;
    E0461 : BOOL ;
    E0462 : BOOL ;
    E0463 : BOOL ;
    E0464 : BOOL ;
    E0465 : BOOL ;	//=CH2_4++ZNE05+HCZ02-QF_10;ALIMENTAÇÃO 24Vdc MOVIFIT +TQ_01;1
    E0466 : BOOL ;	//=CH2_4++ZNE05+HCZ02-QF_20;FONTE DE ALIMENTAÇÃO 440Vac MOVIFIT +TQ_01;1
    E0467 : BOOL ;	//=CH2_4++ZNE05+HCZ02-QF_21;FONTE DE ALIMENTAÇÃO 440Vac OBTURADOR ENTRADA TTS +TQ_01;1
    E0468 : BOOL ;	//=CH2_4++ZNE05+HCZ02-QF_22;FONTE DE ALIMENTAÇÃO 440Vac SAÍDA TTS DO OBTURADOR +TQ_01;1
    E0469 : BOOL ;	//=CH2_4++ZNE05+HCZ02-QF_26;ALIMENTAÇÃO 440Vac ELEVADOR +TQ_01;1
    E0470 : BOOL ;	//=CH2_4++ZNE05+HCZ02-QF_26;FONTE DE ALIMENTAÇÃO 440Vac ELEVADOR BACKUP +TQ_01;1
    E0471 : BOOL ;	//=CH2_4++ZNE05+HCZ02-QF_30;FONTE DE ALIMENTAÇÃO 440Vac MOTOR FREIO DO ELEVADOR +TQ_01;1
    E0472 : BOOL ;	//=CH2_4++ZNE05+HCZ02-QF_31;FREIO DO MOTOR DE BACKUP DO ELEVADOR 440Vac +TQ_01;1
    E0473 : BOOL ;	//=CH2_4++ZNE05+HCZ02-BT_01;SOBRETEMP. RESISTOR DE TRAVAGEM DO ELEVADOR +TQ_01;1
    E0474 : BOOL ;	//=CH2_4++ZNE05+HCZ02-BT_02;SOBRETEMP. RESISTOR DE FRENAGEM DE BACKUP +TQ_01;1
    E0475 : BOOL ;	//=CH2_4++ZNE05+HCZ02-U__01;FALHA MOVIDRIVE +TQ_01;1
    E0476 : BOOL ;	//=CH2_4++ZNE05+HCZ02-U__02;FALHA DE BACKUP DO MOVIDRIVE +TQ_01;1
    E0477 : BOOL ;	//=CH2_4++ZNE05+HCZ02-U__01;ERRO DE COMUNICAÇÃO MOVIDRIVE +TQ_01;1
    E0478 : BOOL ;	//=CH2_4++ZNE05+HCZ02-U__02;BACKUP MOVIDRIVE +TQ_01 ERRO DE COMUNICAÇÃO;1
    E0479 : BOOL ;	//=CH2_4++ZNE05+HCZ02-U__01;EIXO NÃO ZERO MOVIDRIVE +TQ_01;1
    E0480 : BOOL ;	//=CH2_4++ZNE05+HCZ02-U__02;EIXO NÃO ZERO MOVIDRIVE BACKUP +TQ_01;1
    E0481 : BOOL ;	//=CH2_4++ZNE05+HCZ02-KMS02;EFICIÊNCIA DO RELÉ 440Vac +TQ_01;1
    E0482 : BOOL ;	//=CH2_4++ZNE05+HCZ02-KAS02;EFICIÊNCIA DO RELÉ 24Vdc +TQ_01;1
    E0483 : BOOL ;	//=CH2_4++ZNE05+PTZ03-DMC01;FALHA NO MÓDULO ET200S;1
    E0484 : BOOL ;	//=CH2_4++ZNE05+PRE01-DMC01;FALHA NO MÓDULO ET200S;1
    E0485 : BOOL ;	//=CH2_4++ZNE05+HCZ02-QF_23;ALIMENTAÇÃO MAGNETOTÉRMICA 440Vac TRILHA +TTS11 SET06;1
    E0486 : BOOL ;	//=CH2_4++ZNE05+XGA02-SC_01;PORTÃO EM ANOMALIA;1
    E0487 : BOOL ;	//=CH2_4++ZNE05+XGA03-SC_01;PORTÃO EM ANOMALIA;1
    E0488 : BOOL ;
    E0489 : BOOL ;	//=CH2_4++ZNE05+TTS01;CICLO NÃO EM AUTOMÁTICO DA ESTAMPAGEM AUTOMÁTICA;10
    E0490 : BOOL ;	//=CH2_4++ZNE05+TTS01;ANOMALIA DE ESTAMPAGEM AUTOMÁTICA;10
    E0491 : BOOL ;	//=CH2_4++ZNE05+TTS01;EMERGÊNCIA DE ESTAMPAGEM AUTOMÁTICA;10
    E0492 : BOOL ;	//=CH2_4++ZNE05+TTS01;PEQUENO ROBÔ PARA ESTAMPAGEM AUTOMÁTICA;10
    E0493 : BOOL ;	//=CH2_4++ZNE05+TTS01;PEDIDO DE ACESSO DA ESTAMPAGEM AUTOMÁTICA;10
    E0494 : BOOL ;	//=CH2_4++ZNE05+TTS01;AGUARDANDO TRABALHO CONCLUÍDO DA ESTAMPAGEM AUTOMÁTICA;10
    E0495 : BOOL ;	//=CH2_4++ZNE05+TTS01;ESTAÇÃO EXCLUÍDA DA ESTAMPAGEM AUTOMÁTICA;10
    E0496 : BOOL ;	//=CH2_4++ZNE05+TTS01;SETOR NÃO RESTAURADO ESTAMPAGEM AUTOMÁTICA;10
    E0497 : BOOL ;	//=CH2_4++ZNE05+TTS03;CICLO NÃO AUTOMÁTICO DA ESTAMPAGEM DE BACKUP;10
    E0498 : BOOL ;	//=CH2_4++ZNE05+TTS03;ANOMALIA DE ESTAMPA DE BACKUP;10
    E0499 : BOOL ;	//=CH2_4++ZNE05+TTS03;EMERGÊNCIA DE CARIMBO DE BACKUP;10
    E0500 : BOOL ;	//=CH2_4++ZNE05+TTS03;PARCEIRO DO ESPAÇO DE ESTAMPAGEM DE BACKUP;10
    E0501 : BOOL ;	//=CH2_4++ZNE05+TTS03;AGUARDANDO O FIM DO TRABALHO DO BACKUP DE ESTAMPAGEM;10
    E0502 : BOOL ;	//=CH2_4++ZNE05+TTS03;ESTAÇÃO EXCLUÍDA DO BACKUP STAMPING;10
    E0503 : BOOL ;
    E0504 : BOOL ;
    E0505 : BOOL ;	//=CH2_4++ZNE05+TTS06;CICLO DE LIGAÇÃO DE VIDRO NÃO AUTOMÁTICO;10
    E0506 : BOOL ;	//=CH2_4++ZNE05+TTS06;ANOMALIA DE LIGAÇÃO DE VIDRO;10
    E0507 : BOOL ;	//=CH2_4++ZNE05+TTS06;EMERGÊNCIA DE COLAGEM DE VIDRO;10
    E0508 : BOOL ;	//=CH2_4++ZNE05+TTS06;ROBÔ DE JANELA TRASEIRA ESPACIAL PARA COLAGEM DE VIDRO;10
    E0509 : BOOL ;	//=CH2_4++ZNE05+TTS06;PEDIDO DE ACESSO PARA COLAGEM DE VIDRO;10
    E0510 : BOOL ;	//=CH2_4++ZNE05+TTS06;AGUARDANDO A CONCLUSÃO DO TRABALHO DE COLAGEM DE VIDRO;10
    E0511 : BOOL ;	//=CH2_4++ZNE05+TTS06;ESTAÇÃO EXCLUÍDA DA COLAGEM DE VIDRO;10
    E0512 : BOOL ;	//=CH2_4++ZNE05+TTS06;ROBÔ DE PÁRA-BRISA DE COLAGEM DE VIDRO;10
    E0513 : BOOL ;	//=CH2_4++ZNE05+TTS01;SOU PEDIDO DE ACESSO DA ESTAMPAGEM AUTOMÁTICA;14
    E0514 : BOOL ;	//=CH2_4++ZNE05+TTS01;PEDIDO DE ACESSO PM DA ESTAMPAGEM AUTOMÁTICA;13
    E0515 : BOOL ;	//=CH2_4++ZNE05+TTS01;SOU PEDIDO DE ACESSO PARA COLAGEM DE VIDRO;14
    E0516 : BOOL ;	//=CH2_4++ZNE05+TTS01;PEDIDO DE ACESSO PM PARA COLAGEM DE VIDRO;13
    E0517 : BOOL ;	//=CH2_4++ZNE05+TTS06;LUNOTTO - BICO DA COLA DANIFICADO AM;14
    E0518 : BOOL ;	//=CH2_4++ZNE05+TTS06;PARA-BRISA - BICO DA COLA DANIFICADO AM;14
    E0519 : BOOL ;
    E0520 : BOOL ;
    E0521 : BOOL ;
    E0522 : BOOL ;
    E0523 : BOOL ;
    E0524 : BOOL ;
    E0525 : BOOL ;
    E0526 : BOOL ;
    E0527 : BOOL ;
    E0528 : BOOL ;
    E0529 : BOOL ;	//=CH2_4++ZNE05+PTZ03-SB_07;BOTÃO DE EMERGENCIA APERTADO;2
    E0530 : BOOL ;	//=CH2_4++ZNE05+PTZ03-SB_07;EMERGÊNCIA NÃO RESTAURADA;2
    E0531 : BOOL ;	//=CH2_4++ZNE05+PRE01-SB_07;BOTÃO DE EMERGENCIA APERTADO;2
    E0532 : BOOL ;	//=CH2_4++ZNE05+PRE01-SB_07;EMERGÊNCIA NÃO RESTAURADA;2
    E0533 : BOOL ;	//=CH2_4++ZNE05+XGA02-SC_01;MANUTENÇÃO NÃO AGENDADA DE ACESSO ABERTO (GM);2
    E0534 : BOOL ;	//=CH2_4++ZNE05+XGA02-SC_01;ACESSO NÃO RESTAURADO MANUTENÇÃO NÃO PROGRAMADA (GM);2
    E0535 : BOOL ;	//=CH2_4++ZNE05+XGA03-SC_01;MANUTENÇÃO NÃO AGENDADA DE ACESSO ABERTO (GM);2
    E0536 : BOOL ;	//=CH2_4++ZNE05+XGA03-SC_01;ACESSO NÃO RESTAURADO MANUTENÇÃO NÃO PROGRAMADA (GM);2
    E0537 : BOOL ;	//=CH2_4++ZNE05+PRB02-VT_02;BARREIRA INTERDITADA;2
    E0538 : BOOL ;	//=CH2_4++ZNE05+PRB02-VT_02;BARREIRA NÃO RESTAURADA;2
    E0539 : BOOL ;	//=CH2_4++ZNE05+PRB02-BR_04;BARREIRA DE MUTING ENGAJADA;2
    E0540 : BOOL ;	//=CH2_4++ZNE05+PRB02-BR_04;BARREIRA DE MUTING NÃO RESTAURADA;2
    E0541 : BOOL ;
    E0542 : BOOL ;
    E0543 : BOOL ;
    E0544 : BOOL ;
    E0545 : BOOL ;
    E0546 : BOOL ;
    E0547 : BOOL ;
    E0548 : BOOL ;
    E0549 : BOOL ;
    E0550 : BOOL ;
    E0551 : BOOL ;
    E0552 : BOOL ;
    E0553 : BOOL ;	//=CH2_4++ZNE05+XGA02-SC_01;MANUTENÇÃO PROGRAMADA DE ACESSO ABERTO (PM);13
    E0554 : BOOL ;	//=CH2_4++ZNE05+XGA02-SC_01;LIMPEZA TÉCNICA DE ACESSO ABERTO (AM);14
    E0555 : BOOL ;	//=CH2_4++ZNE05+XGA02-SC_01;ACESSO NÃO RESTAURADO PROG. DE MANUTENÇÃO (PM);13
    E0556 : BOOL ;	//=CH2_4++ZNE05+XGA02-SC_01;ACESSO NÃO RESTAURADO LIMPEZA TÉCNICA (AM);14
    E0557 : BOOL ;	//=CH2_4++ZNE05+XGA03-SC_01;MANUTENÇÃO PROGRAMADA DE ACESSO ABERTO (PM);13
    E0558 : BOOL ;	//=CH2_4++ZNE05+XGA03-SC_01;LIMPEZA TÉCNICA DE ACESSO ABERTO (AM);14
    E0559 : BOOL ;	//=CH2_4++ZNE05+XGA03-SC_01;ACESSO NÃO RESTAURADO PROG. DE MANUTENÇÃO (PM);13
    E0560 : BOOL ;	//=CH2_4++ZNE05+XGA03-SC_01;ACESSO NÃO RESTAURADO LIMPEZA TÉCNICA (AM);14
    E0561 : BOOL ;
    E0562 : BOOL ;
    E0563 : BOOL ;
    E0564 : BOOL ;
    E0565 : BOOL ;
    E0566 : BOOL ;
    E0567 : BOOL ;
    E0568 : BOOL ;
    E0569 : BOOL ;
    E0570 : BOOL ;
    E0571 : BOOL ;
    E0572 : BOOL ;
    E0573 : BOOL ;
    E0574 : BOOL ;
    E0575 : BOOL ;
    E0576 : BOOL ;
    E0577 : BOOL ;	//=CH2_4++ZNE05+HCZ02-QF_03;FONTE DE ALIMENTAÇÃO MAGNETOTÉRMICA PARA AR CONDICIONADO 400V;58
    E0578 : BOOL ;	//=CH2_4++ZNE05+HCZ02-QF_15;MAGNETO. PODER PAINEL OPERADOR 24Vdc +PTZ03;58
    E0579 : BOOL ;	//=CH2_4++ZNE05+HCZ02-QF_16;MAGNETO. PODER PAINEL OPERADOR 24Vdc +PRE01;58
    E0580 : BOOL ;	//=CH2_4++ZNE05+HCZ02-U__01;PRÉ-ALARME MOVIDRIVE +TQ_01;58
    E0581 : BOOL ;	//=CH2_4++ZNE05+HCZ02-U__02;PRÉ-ALARME DE BACKUP DO MOVIDRIVE +TQ_01;58
    E0582 : BOOL ;	//=CH2_4++ZNE05+PTZ03-DSP01;PRÉ-ALARME SEM PLC <-> COMUNICAÇÃO IHM;58
    E0583 : BOOL ;	//=CH2_4++ZNE05+PRE01-DSP01;PRÉ-ALARME SEM PLC <-> COMUNICAÇÃO IHM;58
    E0584 : BOOL ;	//=CH2_4++ZNE05+PTZ03-SA_03;PEDIDO DE ACESSO PARA MANUTENÇÃO PLANEJADA (PM);58
    E0585 : BOOL ;	//=CH2_4++ZNE05+PTZ03-SA_03;SOLICITAR ACESSO PARA LIMPEZA TÉCNICA (AM);58
    E0586 : BOOL ;	//=CH2_4++ZNE05+PRE01-SA_03;PEDIDO DE ACESSO PARA MANUTENÇÃO PLANEJADA (PM);58
    E0587 : BOOL ;	//=CH2_4++ZNE05+PRE01-SA_03;SOLICITAR ACESSO PARA LIMPEZA TÉCNICA (AM);58
    E0588 : BOOL ;	//=CH2_4++ZNE05+PTZ03-SA_03;SOLICITAR ACESSO PARA MANUTENÇÃO NÃO PROGRAMADA (GM);58
    E0589 : BOOL ;	//=CH2_4++ZNE05+PRE01-SA_03;SOLICITAR ACESSO PARA MANUTENÇÃO NÃO PROGRAMADA (GM);58
    E0590 : BOOL ;	//=CH2_4++ZNE05+HCZ02-ST_01;CONTROLE DE TEMPERATURA DO GABINETE;58
    E0591 : BOOL ;
    E0592 : BOOL ;
    E0593 : BOOL ;	//=CH2_4++ZNE05+LMN01-DSP01;LINHA PARADA OPERADOR DE LIMO 01 ESTAÇÃO 82 SX;11
    E0594 : BOOL ;	//=CH2_4++ZNE05+LMN03-DSP01;STOP LINE CH.OPERADOR LIMO 03 ESTAÇÃO 83 SX;11
    E0595 : BOOL ;	//=CH2_4++ZNE05+LMN05-DSP01;STOP OPERADOR DE LINHA LIMO 05 ESTAÇÃO 84 SX;11
    E0596 : BOOL ;	//=CH2_4++ZNE05+LMN07-DSP01;STOP OPERADOR DE LINHA LIMO 07 ESTAÇÃO 85 SX;11
    E0597 : BOOL ;	//=CH2_4++ZNE05+LMN09-DSP01;LINHA PARADA OPERADOR DE LIMO 09 ESTAÇÃO 86 SX;11
    E0598 : BOOL ;	//=CH2_4++ZNE05+LMN11-DSP01;LINHA PARADA OPERADOR DE LIMO 11 ESTAÇÃO 83A ESQUERDA;11
    E0599 : BOOL ;
    E0600 : BOOL ;
    E0601 : BOOL ;	//=CH2_4++ZNE05+LMN02-DSP01;STOP OPERADOR DE LINHA LIMO 02 ESTAÇÃO 82 DX;11
    E0602 : BOOL ;	//=CH2_4++ZNE05+LMN04-DSP01;STOP OPERADOR DE LINHA LIMO 04 ESTAÇÃO 83 DX;11
    E0603 : BOOL ;	//=CH2_4++ZNE05+LMN06-DSP01;STOP OPERADOR DE LINHA LIMO 06 ESTAÇÃO 84 DX;11
    E0604 : BOOL ;	//=CH2_4++ZNE05+LMN08-DSP01;STOP OPERADOR DE LINHA LIMO 08 ESTAÇÃO 85 DX;11
    E0605 : BOOL ;	//=CH2_4++ZNE05+LMN10-DSP01;STOP LINE OPERADOR LIMO 10 ESTAÇÃO 86 DX;11
    E0606 : BOOL ;	//=CH2_4++ZNE05+LMN12-DSP01;ESTAÇÃO DE PARADA DA LINHA DO OPERADOR LIMO 12 83A DIREITA;11
    E0607 : BOOL ;
    E0608 : BOOL ;
    E0609 : BOOL ;
    E0610 : BOOL ;
    E0611 : BOOL ;
    E0612 : BOOL ;
    E0613 : BOOL ;
    E0614 : BOOL ;
    E0615 : BOOL ;
    E0616 : BOOL ;
    E0617 : BOOL ;
    E0618 : BOOL ;
    E0619 : BOOL ;
    E0620 : BOOL ;
    E0621 : BOOL ;
    E0622 : BOOL ;
    E0623 : BOOL ;
    E0624 : BOOL ;
    E0625 : BOOL ;	//=CH2_4++ZNE05+ESB03-SQA01;FALHA NO INTERRUPTOR DE LIMITE DE PARAGEM INFERIOR DA PLATAFORMA MÓVEL +ESB;1
    E0626 : BOOL ;	//=CH2_4++ZNE05+ESB03-SQB01;FALHA NO INTERRUPTOR DE LIMITE DE PARADA ALTA DA PLATAFORMA MÓVEL +ESB;1
    E0627 : BOOL ;
    E0628 : BOOL ;
    E0629 : BOOL ;	//=CH2_4++ZNE05+ESB03-SQA01;TIME OUT DESCIDA +ESB;1
    E0630 : BOOL ;	//=CH2_4++ZNE05+ESB03-SQB01;TIME OUT RISE +ESB;1
    E0631 : BOOL ;
    E0632 : BOOL ;
    E0633 : BOOL ;	//=CH2_4++ZNE05+ESB03-HKM03;SONDA TÉRMICA DO MOTOR +ESB;1
    E0634 : BOOL ;
    E0635 : BOOL ;
    E0636 : BOOL ;
    E0637 : BOOL ;
    E0638 : BOOL ;
    E0639 : BOOL ;
    E0640 : BOOL ;
    E0641 : BOOL ;	//=CH2_4++ZNE05+ESB03;ESTAÇÃO EXCLUÍDA PRÉ-ALARME;58
    E0642 : BOOL ;
    E0643 : BOOL ;
    E0644 : BOOL ;
    E0645 : BOOL ;
    E0646 : BOOL ;
    E0647 : BOOL ;
    E0648 : BOOL ;
    E0649 : BOOL ;	//=CH2_4++ZNE05+ESB03;PRÉ-ALARME DE BYPASS DE FALHA ATIVO;58
    E0650 : BOOL ;
    E0651 : BOOL ;
    E0652 : BOOL ;
    E0653 : BOOL ;
    E0654 : BOOL ;
    E0655 : BOOL ;
    E0656 : BOOL ;
    E0657 : BOOL ;	//=CH2_4++ZNE05;EM PRODUÇÃO;19
    E0658 : BOOL ;	//=CH2_4++ZNE05+PTZ03-SB_05;INICIAR CICLO AUTOMÁTICO;15
    E0659 : BOOL ;	//=CH2_4++ZNE05+PRE01-SB_05;INICIAR CICLO AUTOMÁTICO;15
    E0660 : BOOL ;	//=CH2_4++ZNE05+PTZ03-SA_01;CICLO MANUAL SELECIONADO;16
    E0661 : BOOL ;	//=CH2_4++ZNE05+PRE01-SA_01;CICLO MANUAL SELECIONADO;16
    E0662 : BOOL ;	//=CH2_4++ZNE05+PTZ03-SB_04;PARADA DO CICLO;17
    E0663 : BOOL ;	//=CH2_4++ZNE05+PRE01-SB_04;PARADA DO CICLO;17
    E0664 : BOOL ;
    E0665 : BOOL ;
    E0666 : BOOL ;
    E0667 : BOOL ;
    E0668 : BOOL ;
    E0669 : BOOL ;
    E0670 : BOOL ;
    E0671 : BOOL ;
    E0672 : BOOL ;
    E0673 : BOOL ;	//=CH2_4++ZNE05+TTS05-SQA01;FALHA NO INTERRUPTOR DE LIMITE DE PARADA;1
    E0674 : BOOL ;	//=CH2_4++ZNE05+TTS05-SQS01;FALHA NO INTERRUPTOR DE LIMITE DE LENTAÇÃO;1
    E0675 : BOOL ;	//=CH2_4++ZNE05+TTS05-SQC01;FALHA NO INTERRUPTOR DE LIMITE DE CONTROLE DE POSIÇÃO;1
    E0676 : BOOL ;	//=CH2_4++ZNE05+TTS05-B__01;FALHA DA FOTOCÉLULA NA PRESENÇA DO VEÍCULO;1
    E0677 : BOOL ;	//=CH2_4++ZNE05+TTS05;SAIR DO TEMPO DE TRANSFERÊNCIA;1
    E0678 : BOOL ;	//=CH2_4++ZNE05+TTS05;CTRL ENGRENAGEM TTS ANTERIOR;1
    E0679 : BOOL ;	//=CH2_4++ZNE05+TTS05;CTRL ENGRENAGEM PRÓXIMO TTS;1
    E0680 : BOOL ;	//=CH2_4++ZNE05+TTS05;POSIÇÃO CTRL;1
    E0681 : BOOL ;	//=CH2_4++ZNE05+TTS05-M__01;FALHA NO INVERSOR;1
    E0682 : BOOL ;	//=CH2_4++ZNE05+TTS05-M__01;ERRO DE COMUNICAÇÃO DO INVERSOR;1
    E0683 : BOOL ;	//=CH2_4++ZNE05+TTS05-SQA02;FALHA DO INTERRUPTOR DE LIMITE DE PROTEÇÃO QUEDA TRABALHO FECHADO;1
    E0684 : BOOL ;	//=CH2_4++ZNE05+TTS05-SQB02;FALHA DE RESTO ABERTO DO INTERRUPTOR DE LIMITE DE PROTEÇÃO QUEDA;1
    E0685 : BOOL ;	//=CH2_4++ZNE05+TTS05-SQ_01;QUEBRA DA CORREIA DE TRANSMISSÃO TTS;1
    E0686 : BOOL ;	//=CH2_4++ZNE05+TTS05;PRÉ-ALARME DE BYPASS DE FALHA ATIVO;58
    E0687 : BOOL ;	//=CH2_4++ZNE05+TTS05-M__01;PRÉ-ALARME DE CORRENTE ABSORVIDA;58
    E0688 : BOOL ;	//=CH2_4++ZNE05+TTS05-M__01;PRÉ-ALARME DO INVERSOR MOVIMOT;58
    E0689 : BOOL ;	//=CH2_4++ZNE05+TTS05-U__01;ERRO DE COMUNICAÇÃO MOVIFIT;1
    E0690 : BOOL ;	//=CH2_4++ZNE05+TTS05-U__01;INTERRUPTOR MOVIFIT ABERTO 380V;1
    E0691 : BOOL ;	//=CH2_4++ZNE05+TTS05-U__01;AUSÊNCIAS 24 VOLTS MOVIFIT SEGURANÇA;1
    E0692 : BOOL ;	//=CH2_4++ZNE05+TTS05-U__01;AUSÊNCIAS MOVIFIT 24 VOLT;1
    E0693 : BOOL ;	//=CH2_4++ZNE05+TTS05-U__01;ANOMALIA MOVIFIT;1
    E0694 : BOOL ;	//=CH2_4++ZNE05+TTS05-U__01;SOBRECARGA DE TENSÃO DE SAÍDA 0 MOVIFIT;1
    E0695 : BOOL ;	//=CH2_4++ZNE05+TTS05-U__01;TENSÃO DE SAÍDA DE SOBRECARGA SAÍDA 1 MOVIFIT;1
    E0696 : BOOL ;	//=CH2_4++ZNE05+TTS05-U__01;SOBRECARGA DE TENSÃO DO MOVIFIT NA SAÍDA 2;1
    E0697 : BOOL ;	//=CH2_4++ZNE05+TTS05-U__01;SOBRECARGA DE TENSÃO DE SAÍDA 3 MOVIFIT;1
    E0698 : BOOL ;	//=CH2_4++ZNE05+TTS05-U__01;SOBRECARGA DE TENSÃO DO SENSOR MOVIFIT GRUPO 1;1
    E0699 : BOOL ;	//=CH2_4++ZNE05+TTS05-U__01;SOBRECARGA DE TENSÃO DO SENSOR MOVIFIT GRUPO 2;1
    E0700 : BOOL ;	//=CH2_4++ZNE05+TTS05-U__01;SOBRECARGA DE TENSÃO DO SENSOR MOVIFIT GRUPO 3;1
    E0701 : BOOL ;	//=CH2_4++ZNE05+TTS05-U__01;SOBRECARGA DE TENSÃO DO SENSOR MOVIFIT GRUPO 4;1
    E0702 : BOOL ;
    E0703 : BOOL ;
    E0704 : BOOL ;
    E0705 : BOOL ;	//=CH2_4++ZNE05+TTS06-SQA01;FALHA NO INTERRUPTOR DE LIMITE DE PARADA;1
    E0706 : BOOL ;	//=CH2_4++ZNE05+TTS06-SQS01;FALHA NO INTERRUPTOR DE LIMITE DE LENTAÇÃO;1
    E0707 : BOOL ;	//=CH2_4++ZNE05+TTS06-SQC01;FALHA NO INTERRUPTOR DE LIMITE DE CONTROLE DE POSIÇÃO;1
    E0708 : BOOL ;	//=CH2_4++ZNE05+TTS06-B__01;FALHA DA FOTOCÉLULA NA PRESENÇA DO VEÍCULO;1
    E0709 : BOOL ;	//=CH2_4++ZNE05+TTS06;SAIR DO TEMPO DE TRANSFERÊNCIA;1
    E0710 : BOOL ;	//=CH2_4++ZNE05+TTS06;CTRL ENGRENAGEM TTS ANTERIOR;1
    E0711 : BOOL ;	//=CH2_4++ZNE05+TTS06;CTRL ENGRENAGEM PRÓXIMO TTS;1
    E0712 : BOOL ;	//=CH2_4++ZNE05+TTS06;POSIÇÃO CTRL;1
    E0713 : BOOL ;	//=CH2_4++ZNE05+TTS06-M__01;FALHA NO INVERSOR;1
    E0714 : BOOL ;	//=CH2_4++ZNE05+TTS06-M__01;ERRO DE COMUNICAÇÃO DO INVERSOR;1
    E0715 : BOOL ;	//=CH2_4++ZNE05+TTS06-SQA02;FALHA DO INTERRUPTOR DE LIMITE DE PROTEÇÃO QUEDA TRABALHO FECHADO;1
    E0716 : BOOL ;	//=CH2_4++ZNE05+TTS06-SQB02;FALHA DE RESTO ABERTO DO INTERRUPTOR DE LIMITE DE PROTEÇÃO QUEDA;1
    E0717 : BOOL ;	//=CH2_4++ZNE05+TTS06-SQ_01;QUEBRA DA CORREIA DE TRANSMISSÃO TTS;1
    E0718 : BOOL ;	//=CH2_4++ZNE05+TTS06;PRÉ-ALARME DE BYPASS DE FALHA ATIVO;58
    E0719 : BOOL ;	//=CH2_4++ZNE05+TTS06-M__01;PRÉ-ALARME DE CORRENTE ABSORVIDA;58
    E0720 : BOOL ;	//=CH2_4++ZNE05+TTS06-M__01;PRÉ-ALARME DO INVERSOR MOVIMOT;58
    E0721 : BOOL ;	//=CH2_4++ZNE05+TTS06-U__01;ERRO DE COMUNICAÇÃO MOVIFIT;1
    E0722 : BOOL ;	//=CH2_4++ZNE05+TTS06-U__01;INTERRUPTOR MOVIFIT ABERTO 380V;1
    E0723 : BOOL ;	//=CH2_4++ZNE05+TTS06-U__01;AUSÊNCIAS 24 VOLTS MOVIFIT SEGURANÇA;1
    E0724 : BOOL ;	//=CH2_4++ZNE05+TTS06-U__01;AUSÊNCIAS MOVIFIT 24 VOLT;1
    E0725 : BOOL ;	//=CH2_4++ZNE05+TTS06-U__01;ANOMALIA MOVIFIT;1
    E0726 : BOOL ;	//=CH2_4++ZNE05+TTS06-U__01;SOBRECARGA DE TENSÃO DE SAÍDA 0 MOVIFIT;1
    E0727 : BOOL ;	//=CH2_4++ZNE05+TTS06-U__01;TENSÃO DE SAÍDA DE SOBRECARGA SAÍDA 1 MOVIFIT;1
    E0728 : BOOL ;	//=CH2_4++ZNE05+TTS06-U__01;SOBRECARGA DE TENSÃO DO MOVIFIT NA SAÍDA 2;1
    E0729 : BOOL ;	//=CH2_4++ZNE05+TTS06-U__01;SOBRECARGA DE TENSÃO DE SAÍDA 3 MOVIFIT;1
    E0730 : BOOL ;	//=CH2_4++ZNE05+TTS06-U__01;SOBRECARGA DE TENSÃO DO SENSOR MOVIFIT GRUPO 1;1
    E0731 : BOOL ;	//=CH2_4++ZNE05+TTS06-U__01;SOBRECARGA DE TENSÃO DO SENSOR MOVIFIT GRUPO 2;1
    E0732 : BOOL ;	//=CH2_4++ZNE05+TTS06-U__01;SOBRECARGA DE TENSÃO DO SENSOR MOVIFIT GRUPO 3;1
    E0733 : BOOL ;	//=CH2_4++ZNE05+TTS06-U__01;SOBRECARGA DE TENSÃO DO SENSOR MOVIFIT GRUPO 4;1
    E0734 : BOOL ;
    E0735 : BOOL ;
    E0736 : BOOL ;
    E0737 : BOOL ;	//=CH2_4++ZNE05+ESB02-SQA01;FALHA NO INTERRUPTOR DE LIMITE DE PARAGEM INFERIOR DA PLATAFORMA MÓVEL +ESB;1
    E0738 : BOOL ;	//=CH2_4++ZNE05+ESB02-SQB01;FALHA NO INTERRUPTOR DE LIMITE DE PARADA ALTA DA PLATAFORMA MÓVEL +ESB;1
    E0739 : BOOL ;
    E0740 : BOOL ;
    E0741 : BOOL ;	//=CH2_4++ZNE05+ESB02-SQA01;TIME OUT DESCIDA +ESB;1
    E0742 : BOOL ;	//=CH2_4++ZNE05+ESB02-SQB01;TIME OUT RISE +ESB;1
    E0743 : BOOL ;
    E0744 : BOOL ;
    E0745 : BOOL ;	//=CH2_4++ZNE05+ESB02-HKM03;SONDA TÉRMICA DO MOTOR +ESB;1
    E0746 : BOOL ;
    E0747 : BOOL ;
    E0748 : BOOL ;
    E0749 : BOOL ;
    E0750 : BOOL ;
    E0751 : BOOL ;
    E0752 : BOOL ;
    E0753 : BOOL ;	//=CH2_4++ZNE05+ESB02;ESTAÇÃO EXCLUÍDA PRÉ-ALARME;58
    E0754 : BOOL ;
    E0755 : BOOL ;
    E0756 : BOOL ;
    E0757 : BOOL ;
    E0758 : BOOL ;
    E0759 : BOOL ;
    E0760 : BOOL ;
    E0761 : BOOL ;	//=CH2_4++ZNE05+ESB02;PRÉ-ALARME DE BYPASS DE FALHA ATIVO;58
    E0762 : BOOL ;
    E0763 : BOOL ;
    E0764 : BOOL ;
    E0765 : BOOL ;
    E0766 : BOOL ;
    E0767 : BOOL ;
    E0768 : BOOL ;
    E0769 : BOOL ;	//=CH2_4++ZNE05+TTS07-SQA01;FALHA NO INTERRUPTOR DE LIMITE DE PARADA;1
    E0770 : BOOL ;	//=CH2_4++ZNE05+TTS07-SQS01;FALHA NO INTERRUPTOR DE LIMITE DE LENTAÇÃO;1
    E0771 : BOOL ;	//=CH2_4++ZNE05+TTS07-SQC01;FALHA NO INTERRUPTOR DE LIMITE DE CONTROLE DE POSIÇÃO;1
    E0772 : BOOL ;	//=CH2_4++ZNE05+TTS07-B__01;FALHA DA FOTOCÉLULA NA PRESENÇA DO VEÍCULO;1
    E0773 : BOOL ;	//=CH2_4++ZNE05+TTS07;SAIR DO TEMPO DE TRANSFERÊNCIA;1
    E0774 : BOOL ;	//=CH2_4++ZNE05+TTS07;CTRL ENGRENAGEM TTS ANTERIOR;1
    E0775 : BOOL ;	//=CH2_4++ZNE05+TTS07;CTRL ENGRENAGEM PRÓXIMO TTS;1
    E0776 : BOOL ;	//=CH2_4++ZNE05+TTS07;POSIÇÃO CTRL;1
    E0777 : BOOL ;	//=CH2_4++ZNE05+TTS07-M__01;FALHA NO INVERSOR;1
    E0778 : BOOL ;	//=CH2_4++ZNE05+TTS07-M__01;ERRO DE COMUNICAÇÃO DO INVERSOR;1
    E0779 : BOOL ;	//=CH2_4++ZNE05+TTS07-SQA02;FALHA DO INTERRUPTOR DE LIMITE DE PROTEÇÃO QUEDA TRABALHO FECHADO;1
    E0780 : BOOL ;	//=CH2_4++ZNE05+TTS07-SQB02;FALHA DE RESTO ABERTO DO INTERRUPTOR DE LIMITE DE PROTEÇÃO QUEDA;1
    E0781 : BOOL ;	//=CH2_4++ZNE05+TTS07-SQ_01;QUEBRA DA CORREIA DE TRANSMISSÃO TTS;1
    E0782 : BOOL ;	//=CH2_4++ZNE05+TTS07;PRÉ-ALARME DE BYPASS DE FALHA ATIVO;58
    E0783 : BOOL ;	//=CH2_4++ZNE05+TTS07-M__01;PRÉ-ALARME DE CORRENTE ABSORVIDA;58
    E0784 : BOOL ;	//=CH2_4++ZNE05+TTS07-M__01;PRÉ-ALARME DO INVERSOR MOVIMOT;58
    E0785 : BOOL ;	//=CH2_4++ZNE05+TTS07-U__01;ERRO DE COMUNICAÇÃO MOVIFIT;1
    E0786 : BOOL ;	//=CH2_4++ZNE05+TTS07-U__01;INTERRUPTOR MOVIFIT ABERTO 380V;1
    E0787 : BOOL ;	//=CH2_4++ZNE05+TTS07-U__01;AUSÊNCIAS 24 VOLTS MOVIFIT SEGURANÇA;1
    E0788 : BOOL ;	//=CH2_4++ZNE05+TTS07-U__01;AUSÊNCIAS MOVIFIT 24 VOLT;1
    E0789 : BOOL ;	//=CH2_4++ZNE05+TTS07-U__01;ANOMALIA MOVIFIT MOVIFIT;1
    E0790 : BOOL ;	//=CH2_4++ZNE05+TTS07-U__01;SOBRECARGA DE TENSÃO DE SAÍDA 0 MOVIFIT;1
    E0791 : BOOL ;	//=CH2_4++ZNE05+TTS07-U__01;TENSÃO DE SAÍDA DE SOBRECARGA SAÍDA 1 MOVIFIT;1
    E0792 : BOOL ;	//=CH2_4++ZNE05+TTS07-U__01;SOBRECARGA DE TENSÃO DO MOVIFIT NA SAÍDA 2;1
    E0793 : BOOL ;	//=CH2_4++ZNE05+TTS07-U__01;SOBRECARGA DE TENSÃO DE SAÍDA 3 MOVIFIT;1
    E0794 : BOOL ;	//=CH2_4++ZNE05+TTS07-U__01;SOBRECARGA DE TENSÃO DO SENSOR MOVIFIT GRUPO 1;1
    E0795 : BOOL ;	//=CH2_4++ZNE05+TTS07-U__01;SOBRECARGA DE TENSÃO DO SENSOR MOVIFIT GRUPO 2;1
    E0796 : BOOL ;	//=CH2_4++ZNE05+TTS07-U__01;SOBRECARGA DE TENSÃO DO SENSOR MOVIFIT GRUPO 3;1
    E0797 : BOOL ;	//=CH2_4++ZNE05+TTS07-U__01;SOBRECARGA DE TENSÃO DO SENSOR MOVIFIT GRUPO 4;1
    E0798 : BOOL ;
    E0799 : BOOL ;
    E0800 : BOOL ;
    E0801 : BOOL ;	//=CH2_4++ZNE05+TTS08-SQA01;FALHA NO INTERRUPTOR DE LIMITE DE PARADA;1
    E0802 : BOOL ;	//=CH2_4++ZNE05+TTS08-SQS01;FALHA NO INTERRUPTOR DE LIMITE DE LENTAÇÃO;1
    E0803 : BOOL ;	//=CH2_4++ZNE05+TTS08-SQC01;FALHA NO INTERRUPTOR DE LIMITE DE CONTROLE DE POSIÇÃO;1
    E0804 : BOOL ;	//=CH2_4++ZNE05+TTS08-B__01;FALHA DA FOTOCÉLULA NA PRESENÇA DO VEÍCULO;1
    E0805 : BOOL ;	//=CH2_4++ZNE05+TTS08;SAIR DO TEMPO DE TRANSFERÊNCIA;1
    E0806 : BOOL ;	//=CH2_4++ZNE05+TTS08;CTRL ENGRENAGEM TTS ANTERIOR;1
    E0807 : BOOL ;	//=CH2_4++ZNE05+TTS08;CTRL ENGRENAGEM PRÓXIMO TTS;1
    E0808 : BOOL ;	//=CH2_4++ZNE05+TTS08;POSIÇÃO CTRL;1
    E0809 : BOOL ;	//=CH2_4++ZNE05+TTS08-M__01;FALHA NO INVERSOR;1
    E0810 : BOOL ;	//=CH2_4++ZNE05+TTS08-M__01;ERRO DE COMUNICAÇÃO DO INVERSOR;1
    E0811 : BOOL ;	//=CH2_4++ZNE05+TTS08-SQA02;FALHA DO INTERRUPTOR DE LIMITE DE PROTEÇÃO QUEDA TRABALHO FECHADO;1
    E0812 : BOOL ;	//=CH2_4++ZNE05+TTS08-SQB02;FALHA DE RESTO ABERTO DO INTERRUPTOR DE LIMITE DE PROTEÇÃO QUEDA;1
    E0813 : BOOL ;	//=CH2_4++ZNE05+TTS08-SQ_01;QUEBRA DA CORREIA DE TRANSMISSÃO TTS;1
    E0814 : BOOL ;	//=CH2_4++ZNE05+TTS08;PRÉ-ALARME DE BYPASS DE FALHA ATIVO;58
    E0815 : BOOL ;	//=CH2_4++ZNE05+TTS08-M__01;PRÉ-ALARME DE CORRENTE ABSORVIDA;58
    E0816 : BOOL ;	//=CH2_4++ZNE05+TTS08-M__01;PRÉ-ALARME DO INVERSOR MOVIMOT;58
    E0817 : BOOL ;	//=CH2_4++ZNE05+TTS08-U__01;ERRO DE COMUNICAÇÃO MOVIFIT;1
    E0818 : BOOL ;	//=CH2_4++ZNE05+TTS08-U__01;INTERRUPTOR MOVIFIT ABERTO 380V;1
    E0819 : BOOL ;	//=CH2_4++ZNE05+TTS08-U__01;AUSÊNCIAS 24 VOLTS MOVIFIT SEGURANÇA;1
    E0820 : BOOL ;	//=CH2_4++ZNE05+TTS08-U__01;AUSÊNCIAS MOVIFIT 24 VOLT;1
    E0821 : BOOL ;	//=CH2_4++ZNE05+TTS08-U__01;ANOMALIA MOVIFIT;1
    E0822 : BOOL ;	//=CH2_4++ZNE05+TTS08-U__01;SOBRECARGA DE TENSÃO DE SAÍDA 0 MOVIFIT;1
    E0823 : BOOL ;	//=CH2_4++ZNE05+TTS08-U__01;TENSÃO DE SAÍDA DE SOBRECARGA SAÍDA 1 MOVIFIT;1
    E0824 : BOOL ;	//=CH2_4++ZNE05+TTS08-U__01;SOBRECARGA DE TENSÃO DO MOVIFIT NA SAÍDA 2;1
    E0825 : BOOL ;	//=CH2_4++ZNE05+TTS08-U__01;SOBRECARGA DE TENSÃO DE SAÍDA 3 MOVIFIT;1
    E0826 : BOOL ;	//=CH2_4++ZNE05+TTS08-U__01;SOBRECARGA DE TENSÃO DO SENSOR MOVIFIT GRUPO 1;1
    E0827 : BOOL ;	//=CH2_4++ZNE05+TTS08-U__01;SOBRECARGA DE TENSÃO DO SENSOR MOVIFIT GRUPO 2;1
    E0828 : BOOL ;	//=CH2_4++ZNE05+TTS08-U__01;SOBRECARGA DE TENSÃO DO SENSOR MOVIFIT GRUPO 3;1
    E0829 : BOOL ;	//=CH2_4++ZNE05+TTS08-U__01;SOBRECARGA DE TENSÃO DO SENSOR MOVIFIT GRUPO 4;1
    E0830 : BOOL ;
    E0831 : BOOL ;
    E0832 : BOOL ;
    E0833 : BOOL ;	//=CH2_4++ZNE05+TTS09-SQA01;FALHA NO INTERRUPTOR DE LIMITE DE PARADA;1
    E0834 : BOOL ;	//=CH2_4++ZNE05+TTS09-SQS01;FALHA NO INTERRUPTOR DE LIMITE DE LENTAÇÃO;1
    E0835 : BOOL ;	//=CH2_4++ZNE05+TTS09-SQC01;FALHA NO INTERRUPTOR DE LIMITE DE CONTROLE DE POSIÇÃO;1
    E0836 : BOOL ;	//=CH2_4++ZNE05+TTS09-B__01;FALHA DA FOTOCÉLULA NA PRESENÇA DO VEÍCULO;1
    E0837 : BOOL ;	//=CH2_4++ZNE05+TTS09;SAIR DO TEMPO DE TRANSFERÊNCIA;1
    E0838 : BOOL ;	//=CH2_4++ZNE05+TTS09;CTRL ENGRENAGEM TTS ANTERIOR;1
    E0839 : BOOL ;	//=CH2_4++ZNE05+TTS09;CTRL ENGRENAGEM PRÓXIMO TTS;1
    E0840 : BOOL ;	//=CH2_4++ZNE05+TTS09;POSIÇÃO CTRL;1
    E0841 : BOOL ;	//=CH2_4++ZNE05+TTS09-M__01;FALHA NO INVERSOR;1
    E0842 : BOOL ;	//=CH2_4++ZNE05+TTS09-M__01;ERRO DE COMUNICAÇÃO DO INVERSOR;1
    E0843 : BOOL ;	//=CH2_4++ZNE05+TTS09-SQA02;FALHA DO INTERRUPTOR DE LIMITE DE PROTEÇÃO QUEDA TRABALHO FECHADO;1
    E0844 : BOOL ;	//=CH2_4++ZNE05+TTS09-SQB02;FALHA DE RESTO ABERTO DO INTERRUPTOR DE LIMITE DE PROTEÇÃO QUEDA;1
    E0845 : BOOL ;	//=CH2_4++ZNE05+TTS09-SQ_01;QUEBRA DA CORREIA DE TRANSMISSÃO TTS;1
    E0846 : BOOL ;	//=CH2_4++ZNE05+TTS09;PRÉ-ALARME DE BYPASS DE FALHA ATIVO;58
    E0847 : BOOL ;	//=CH2_4++ZNE05+TTS09-M__01;PRÉ-ALARME DE CORRENTE ABSORVIDA;58
    E0848 : BOOL ;	//=CH2_4++ZNE05+TTS09-M__01;PRÉ-ALARME DO INVERSOR MOVIMOT;58
    E0849 : BOOL ;	//=CH2_4++ZNE05+TTS09-U__01;ERRO DE COMUNICAÇÃO MOVIFIT;1
    E0850 : BOOL ;	//=CH2_4++ZNE05+TTS09-U__01;INTERRUPTOR MOVIFIT ABERTO 380V;1
    E0851 : BOOL ;	//=CH2_4++ZNE05+TTS09-U__01;AUSÊNCIAS 24 VOLTS MOVIFIT SEGURANÇA;1
    E0852 : BOOL ;	//=CH2_4++ZNE05+TTS09-U__01;AUSÊNCIAS MOVIFIT 24 VOLT;1
    E0853 : BOOL ;	//=CH2_4++ZNE05+TTS09-U__01;ANOMALIA MOVIFIT;1
    E0854 : BOOL ;	//=CH2_4++ZNE05+TTS09-U__01;SOBRECARGA DE TENSÃO DE SAÍDA 0 MOVIFIT;1
    E0855 : BOOL ;	//=CH2_4++ZNE05+TTS09-U__01;TENSÃO DE SAÍDA DE SOBRECARGA SAÍDA 1 MOVIFIT;1
    E0856 : BOOL ;	//=CH2_4++ZNE05+TTS09-U__01;SOBRECARGA DE TENSÃO DO MOVIFIT NA SAÍDA 2;1
    E0857 : BOOL ;	//=CH2_4++ZNE05+TTS09-U__01;SOBRECARGA DE TENSÃO DE SAÍDA 3 MOVIFIT;1
    E0858 : BOOL ;	//=CH2_4++ZNE05+TTS09-U__01;SOBRECARGA DE TENSÃO DO SENSOR MOVIFIT GRUPO 1;1
    E0859 : BOOL ;	//=CH2_4++ZNE05+TTS09-U__01;SOBRECARGA DE TENSÃO DO SENSOR MOVIFIT GRUPO 2;1
    E0860 : BOOL ;	//=CH2_4++ZNE05+TTS09-U__01;SOBRECARGA DE TENSÃO DO SENSOR MOVIFIT GRUPO 3;1
    E0861 : BOOL ;	//=CH2_4++ZNE05+TTS09-U__01;SOBRECARGA DE TENSÃO DO SENSOR MOVIFIT GRUPO 4;1
    E0862 : BOOL ;
    E0863 : BOOL ;
    E0864 : BOOL ;
    E0865 : BOOL ;	//=CH2_4++ZNE05+TTS10-SQA01;FALHA NO INTERRUPTOR DE LIMITE DE PARADA;1
    E0866 : BOOL ;	//=CH2_4++ZNE05+TTS10-SQS01;FALHA NO INTERRUPTOR DE LIMITE DE LENTAÇÃO;1
    E0867 : BOOL ;	//=CH2_4++ZNE05+TTS10-SQC01;FALHA NO INTERRUPTOR DE LIMITE DE CONTROLE DE POSIÇÃO;1
    E0868 : BOOL ;	//=CH2_4++ZNE05+TTS10-B__01;FALHA DA FOTOCÉLULA NA PRESENÇA DO VEÍCULO;1
    E0869 : BOOL ;	//=CH2_4++ZNE05+TTS10;SAIR DO TEMPO DE TRANSFERÊNCIA;1
    E0870 : BOOL ;	//=CH2_4++ZNE05+TTS10;CTRL ENGRENAGEM TTS ANTERIOR;1
    E0871 : BOOL ;	//=CH2_4++ZNE05+TTS10;CTRL ENGRENAGEM PRÓXIMO TTS;1
    E0872 : BOOL ;	//=CH2_4++ZNE05+TTS10;POSIÇÃO CTRL;1
    E0873 : BOOL ;	//=CH2_4++ZNE05+TTS10-M__01;FALHA NO INVERSOR;1
    E0874 : BOOL ;	//=CH2_4++ZNE05+TTS10-M__01;ERRO DE COMUNICAÇÃO DO INVERSOR;1
    E0875 : BOOL ;	//=CH2_4++ZNE05+TTS10-SQA02;FALHA DO INTERRUPTOR DE LIMITE DE PROTEÇÃO QUEDA TRABALHO FECHADO;1
    E0876 : BOOL ;	//=CH2_4++ZNE05+TTS10-SQB02;FALHA DE RESTO ABERTO DO INTERRUPTOR DE LIMITE DE PROTEÇÃO QUEDA;1
    E0877 : BOOL ;	//=CH2_4++ZNE05+TTS10-SQ_01;QUEBRA DA CORREIA DE TRANSMISSÃO TTS;1
    E0878 : BOOL ;	//=CH2_4++ZNE05+TTS10;PRÉ-ALARME DE BYPASS DE FALHA ATIVO;58
    E0879 : BOOL ;	//=CH2_4++ZNE05+TTS10-M__01;PRÉ-ALARME DE CORRENTE ABSORVIDA;58
    E0880 : BOOL ;	//=CH2_4++ZNE05+TTS10-M__01;PRÉ-ALARME DO INVERSOR MOVIMOT;58
    E0881 : BOOL ;	//=CH2_4++ZNE05+TTS10-U__01;ERRO DE COMUNICAÇÃO MOVIFIT;1
    E0882 : BOOL ;	//=CH2_4++ZNE05+TTS10-U__01;INTERRUPTOR MOVIFIT ABERTO 380V;1
    E0883 : BOOL ;	//=CH2_4++ZNE05+TTS10-U__01;AUSÊNCIAS 24 VOLTS MOVIFIT SEGURANÇA;1
    E0884 : BOOL ;	//=CH2_4++ZNE05+TTS10-U__01;AUSÊNCIAS MOVIFIT 24 VOLT;1
    E0885 : BOOL ;	//=CH2_4++ZNE05+TTS10-U__01;ANOMALIA MOVIFIT;1
    E0886 : BOOL ;	//=CH2_4++ZNE05+TTS10-U__01;SOBRECARGA DE TENSÃO DE SAÍDA 0 MOVIFIT;1
    E0887 : BOOL ;	//=CH2_4++ZNE05+TTS10-U__01;TENSÃO DE SAÍDA DE SOBRECARGA SAÍDA 1 MOVIFIT;1
    E0888 : BOOL ;	//=CH2_4++ZNE05+TTS10-U__01;SOBRECARGA DE TENSÃO DO MOVIFIT NA SAÍDA 2;1
    E0889 : BOOL ;	//=CH2_4++ZNE05+TTS10-U__01;SOBRECARGA DE TENSÃO DE SAÍDA 3 MOVIFIT;1
    E0890 : BOOL ;	//=CH2_4++ZNE05+TTS10-U__01;SOBRECARGA DE TENSÃO DO SENSOR MOVIFIT GRUPO 1;1
    E0891 : BOOL ;	//=CH2_4++ZNE05+TTS10-U__01;SOBRECARGA DE TENSÃO DO SENSOR MOVIFIT GRUPO 2;1
    E0892 : BOOL ;	//=CH2_4++ZNE05+TTS10-U__01;SOBRECARGA DE TENSÃO DO SENSOR MOVIFIT GRUPO 3;1
    E0893 : BOOL ;	//=CH2_4++ZNE05+TTS10-U__01;SOBRECARGA DE TENSÃO DO SENSOR MOVIFIT GRUPO 4;1
    E0894 : BOOL ;
    E0895 : BOOL ;
    E0896 : BOOL ;
    E0897 : BOOL ;	//=CH2_4++ZNE05+TTS11-SQA01;FALHA NO INTERRUPTOR DE LIMITE DE PARADA;1
    E0898 : BOOL ;	//=CH2_4++ZNE05+TTS11-SQS01;FALHA NO INTERRUPTOR DE LIMITE DE LENTAÇÃO;1
    E0899 : BOOL ;	//=CH2_4++ZNE05+TTS11-SQC01;FALHA NO INTERRUPTOR DE LIMITE DE CONTROLE DE POSIÇÃO;1
    E0900 : BOOL ;	//=CH2_4++ZNE05+TTS11-B__01;FALHA DA FOTOCÉLULA NA PRESENÇA DO VEÍCULO;1
    E0901 : BOOL ;	//=CH2_4++ZNE05+TTS11;SAIR DO TEMPO DE TRANSFERÊNCIA;1
    E0902 : BOOL ;	//=CH2_4++ZNE05+TTS11;CTRL ENGRENAGEM TTS ANTERIOR;1
    E0903 : BOOL ;	//=CH2_4++ZNE05+TTS11;CTRL ENGRENAGEM PRÓXIMO TTS;1
    E0904 : BOOL ;	//=CH2_4++ZNE05+TTS11;POSIÇÃO CTRL;1
    E0905 : BOOL ;	//=CH2_4++ZNE05+TTS11-M__01;FALHA NO INVERSOR;1
    E0906 : BOOL ;	//=CH2_4++ZNE05+TTS11-M__01;ERRO DE COMUNICAÇÃO DO INVERSOR;1
    E0907 : BOOL ;	//=CH2_4++ZNE05+TTS11-SQA02;FALHA DO INTERRUPTOR DE LIMITE DE PROTEÇÃO QUEDA TRABALHO FECHADO;1
    E0908 : BOOL ;	//=CH2_4++ZNE05+TTS11-SQB02;FALHA DE RESTO ABERTO DO INTERRUPTOR DE LIMITE DE PROTEÇÃO QUEDA;1
    E0909 : BOOL ;	//=CH2_4++ZNE05+TTS11-SQ_01;QUEBRA DA CORREIA DE TRANSMISSÃO TTS;1
    E0910 : BOOL ;	//=CH2_4++ZNE05+TTS11;PRÉ-ALARME DE BYPASS DE FALHA ATIVO;58
    E0911 : BOOL ;	//=CH2_4++ZNE05+TTS11-M__01;PRÉ-ALARME DE CORRENTE ABSORVIDA;58
    E0912 : BOOL ;	//=CH2_4++ZNE05+TTS11-M__01;PRÉ-ALARME DO INVERSOR MOVIMOT;58
    E0913 : BOOL ;	//=CH2_4++ZNE05+TTS11-U__01;ERRO DE COMUNICAÇÃO MOVIFIT;1
    E0914 : BOOL ;	//=CH2_4++ZNE05+TTS11-U__01;INTERRUPTOR MOVIFIT ABERTO 380V;1
    E0915 : BOOL ;	//=CH2_4++ZNE05+TTS11-U__01;AUSÊNCIAS 24 VOLTS MOVIFIT SEGURANÇA;1
    E0916 : BOOL ;	//=CH2_4++ZNE05+TTS11-U__01;AUSÊNCIAS MOVIFIT 24 VOLT;1
    E0917 : BOOL ;	//=CH2_4++ZNE05+TTS11-U__01;ANOMALIA MOVIFIT;1
    E0918 : BOOL ;	//=CH2_4++ZNE05+TTS11-U__01;SOBRECARGA DE TENSÃO DE SAÍDA 0 MOVIFIT;1
    E0919 : BOOL ;	//=CH2_4++ZNE05+TTS11-U__01;TENSÃO DE SAÍDA DE SOBRECARGA SAÍDA 1 MOVIFIT;1
    E0920 : BOOL ;	//=CH2_4++ZNE05+TTS11-U__01;SOBRECARGA DE TENSÃO DO MOVIFIT NA SAÍDA 2;1
    E0921 : BOOL ;	//=CH2_4++ZNE05+TTS11-U__01;SOBRECARGA DE TENSÃO DE SAÍDA 3 MOVIFIT;1
    E0922 : BOOL ;	//=CH2_4++ZNE05+TTS11-U__01;SOBRECARGA DE TENSÃO DO SENSOR MOVIFIT GRUPO 1;1
    E0923 : BOOL ;	//=CH2_4++ZNE05+TTS11-U__01;SOBRECARGA DE TENSÃO DO SENSOR MOVIFIT GRUPO 2;1
    E0924 : BOOL ;	//=CH2_4++ZNE05+TTS11-U__01;SOBRECARGA DE TENSÃO DO SENSOR MOVIFIT GRUPO 3;1
    E0925 : BOOL ;	//=CH2_4++ZNE05+TTS11-U__01;SOBRECARGA DE TENSÃO DO SENSOR MOVIFIT GRUPO 4;1
    E0926 : BOOL ;
    E0927 : BOOL ;
    E0928 : BOOL ;
    E0929 : BOOL ;	//=CH2_4++ZNE05+TQ_01-SQA02;FALHA NO INTERRUPTOR DE LIMITE DE PARADA;1
    E0930 : BOOL ;	//=CH2_4++ZNE05+TQ_01-SQS01;FALHA NO INTERRUPTOR DE LIMITE DE LENTAÇÃO;1
    E0931 : BOOL ;
    E0932 : BOOL ;
    E0933 : BOOL ;	//=CH2_4++ZNE05+TQ_01;SAIR DO TEMPO DE TRANSFERÊNCIA;1
    E0934 : BOOL ;	//=CH2_4++ZNE05+TQ_01;CTRL ENGRENAGEM TTS ANTERIOR;1
    E0935 : BOOL ;	//=CH2_4++ZNE05+TQ_01;CTRL ENGRENAGEM PRÓXIMO TTS;1
    E0936 : BOOL ;	//=CH2_4++ZNE05+TQ_01;POSIÇÃO CTRL;1
    E0937 : BOOL ;	//=CH2_4++ZNE05+TQ_01-U__01;FALHA MOVIFIT FC/30;1
    E0938 : BOOL ;	//=CH2_4++ZNE05+TQ_01-U__01;COMUNICAÇÃO MOVIFIT FC/30;1
    E0939 : BOOL ;	//=CH2_4++ZNE05+TQ_01-SQ_01;FALHA NO INTERRUPTOR DE LIMITE DE PROTEÇÃO CONTRA QUEDA DE SAÍDA TTS;1
    E0940 : BOOL ;	//=CH2_4++ZNE05+TQ_01-SQ_02;FALHA NO INTERRUPTOR DE LIMITE DE PROTEÇÃO CONTRA QUEDA DE ENTRADA TTS;1
    E0941 : BOOL ;
    E0942 : BOOL ;	//=CH2_4++ZNE05+TQ_01;TTS FAULT BYPASS PRÉ-ALARME ATIVO;58
    E0943 : BOOL ;	//=CH2_4++ZNE05+TQ_01-M__04;PRÉ-ALARME DE TRILHA TTS DE CORRENTE ABSORVIDA;58
    E0944 : BOOL ;	//=CH2_4++ZNE05+TQ_01-M__04;PRÉ-ALARME MOVIFIT NA ROTA TTS;58
    E0945 : BOOL ;	//=CH2_4++ZNE05+TQ_01-U__01;ERRO DE COMUNICAÇÃO MOVIFIT;1
    E0946 : BOOL ;	//=CH2_4++ZNE05+TQ_01-U__01;INTERRUPTOR MOVIFIT ABERTO 380V;1
    E0947 : BOOL ;	//=CH2_4++ZNE05+TQ_01-U__01;AUSÊNCIAS 24 VOLTS MOVIFIT SEGURANÇA;1
    E0948 : BOOL ;	//=CH2_4++ZNE05+TQ_01-U__01;AUSÊNCIAS MOVIFIT 24 VOLT;1
    E0949 : BOOL ;	//=CH2_4++ZNE05+TQ_01-U__01;ANOMALIA MOVIFIT;1
    E0950 : BOOL ;	//=CH2_4++ZNE05+TQ_01-U__01;SOBRECARGA DE TENSÃO DE SAÍDA 0 MOVIFIT;1
    E0951 : BOOL ;	//=CH2_4++ZNE05+TQ_01-U__01;TENSÃO DE SAÍDA DE SOBRECARGA SAÍDA 1 MOVIFIT;1
    E0952 : BOOL ;	//=CH2_4++ZNE05+TQ_01-U__01;SOBRECARGA DE TENSÃO DO MOVIFIT NA SAÍDA 2;1
    E0953 : BOOL ;	//=CH2_4++ZNE05+TQ_01-U__01;SOBRECARGA DE TENSÃO DE SAÍDA 3 MOVIFIT;1
    E0954 : BOOL ;	//=CH2_4++ZNE05+TQ_01-U__01;SOBRECARGA DE TENSÃO DO SENSOR MOVIFIT GRUPO 1;1
    E0955 : BOOL ;	//=CH2_4++ZNE05+TQ_01-U__01;SOBRECARGA DE TENSÃO DO SENSOR MOVIFIT GRUPO 2;1
    E0956 : BOOL ;	//=CH2_4++ZNE05+TQ_01-U__01;SOBRECARGA DE TENSÃO DO SENSOR MOVIFIT GRUPO 3;1
    E0957 : BOOL ;	//=CH2_4++ZNE05+TQ_01-U__01;SOBRECARGA DE TENSÃO DO SENSOR MOVIFIT GRUPO 4;1
    E0958 : BOOL ;
    E0959 : BOOL ;
    E0960 : BOOL ;
    E0961 : BOOL ;	//=CH2_4++ZNE05+TQ_01-SQE01;ALTA VIAGEM EXTRA;1
    E0962 : BOOL ;	//=CH2_4++ZNE05+TQ_01-SQE02;BAIXA VIAGEM EXTRA;1
    E0963 : BOOL ;	//=CH2_4++ZNE05+TQ_01-SQC01;FALHA NO INTERRUPTOR DE LIMITE ZERO;1
    E0964 : BOOL ;	//=CH2_4++ZNE05+TQ_01-SQ_01;TRAVA 1 NÃO INSERIDA;1
    E0965 : BOOL ;	//=CH2_4++ZNE05+TQ_01-SQ_02;TRAVA 2 NÃO INSERIDA;1
    E0966 : BOOL ;	//=CH2_4++ZNE05+TQ_01-SQ_03;QUEBRA DA CORREIA;1
    E0967 : BOOL ;	//=CH2_4++ZNE05+TQ_01-SQA01;FALHA FC OBTURADOR DA PARTE MÓVEL DESENGATADO;1
    E0968 : BOOL ;	//=CH2_4++ZNE05+TQ_01-SQB01;FC FALHA PEÇA MÓVEL OBTURADOR INSERIDO;1
    E0969 : BOOL ;	//=CH2_4++ZNE05+TQ_01-SQA03;FALHA FC TTS OBTURADOR DE ENTRADA DESATIVADO;1
    E0970 : BOOL ;	//=CH2_4++ZNE05+TQ_01-SQB03;FALHA FC TTS OBTURADOR DE ENTRADA LIGADO;1
    E0971 : BOOL ;	//=CH2_4++ZNE05+TQ_01-SQA04;FC FALHA TTS OBTURADOR DE SAÍDA DESATIVADO;1
    E0972 : BOOL ;	//=CH2_4++ZNE05+TQ_01-SQB04;FC FALHA TTS OBTURADOR DE SAÍDA LIGADO;1
    E0973 : BOOL ;	//=CH2_4++ZNE05+TQ_01-B__03;FALHA FTC DE PORTA ABERTA +TQ_01;1
    E0974 : BOOL ;	//=CH2_4++ZNE05+TQ_01-SQB05;BUHL01 NÃO DESATIVADO;1
    E0975 : BOOL ;
    E0976 : BOOL ;	//=CH2_4++ZNE05+TQ_01-SQB06;BUHL02 NÃO DESATIVADO;1
    E0977 : BOOL ;	//=CH2_4++ZNE05+TQ_01-B__01;FALHA FTC FORA DA ENTRADA + FOLGA TQ_01;1
    E0978 : BOOL ;	//=CH2_4++ZNE05+TQ_01-B__02;FALHA FTC FORA DA SAÍDA +TQ_01;1
    E0979 : BOOL ;	//=CH2_4++ZNE05+TQ_01-SP_01;PRESSÃO DE AR ??INSUFICIENTE DE BUHL;1
    E0980 : BOOL ;
    E0981 : BOOL ;
    E0982 : BOOL ;	//=CH2_4++ZNE05+TQ_01;ANOMALIA DE SELEÇÃO DE LINHA/BACKUP MOVIDRIVE;1
    E0983 : BOOL ;	//=CH2_4++ZNE05+TQ_01-U__01;FALHA DE OTQ DO MOVIFIT;1
    E0984 : BOOL ;	//=CH2_4++ZNE05+TQ_01-U__01;ERRO DE COMUNICAÇÃO MOVIFIT OTQ;1
    E0985 : BOOL ;	//=CH2_4++ZNE05+TQ_01-SQB01;TEMPO LIMITE DE INSERÇÃO DO OBTURADOR DA PEÇA MÓVEL;1
    E0986 : BOOL ;	//=CH2_4++ZNE05+TQ_01-SQA01;TEMPO LIMITE DE DESENGATE DO OBTURADOR DA PARTE MÓVEL;1
    E0987 : BOOL ;	//=CH2_4++ZNE05+TQ_01-SQB03;FC TIMEOUT TTS ENTRADA OBTURADOR LIGADO;1
    E0988 : BOOL ;	//=CH2_4++ZNE05+TQ_01-SQA03;FC TIMEOUT TTS OBTURADOR DE ENTRADA DESATIVADO;1
    E0989 : BOOL ;	//=CH2_4++ZNE05+TQ_01-SQB04;FC TIMEOUT TTS SAÍDA OBTURADOR LIGADO;1
    E0990 : BOOL ;	//=CH2_4++ZNE05+TQ_01-SQA04;FC TIMEOUT SHUTTER TTS SAÍDA DESATIVADA;1
    E0991 : BOOL ;	//=CH2_4++ZNE05+TQ_01-SE_01;TEMPO LIMITE DE POSIÇÃO ALTA;1
    E0992 : BOOL ;	//=CH2_4++ZNE05+TQ_01-SE_01;TIMEOUT POSIZIONE BASSA ;1
    E0993 : BOOL ;	//=CH2_4++ZNE05+TQ_01-U__01;PRÉ-ALARME MOVIFIT INVERSOR OTQ;58
    E0994 : BOOL ;	//=CH2_4++ZNE05+TQ_01-U__01;PRÉ-ALARME DE CORRENTE ABSORVIDA DO INVERSOR OTQ;58
    E0995 : BOOL ;
    E0996 : BOOL ;
    E0997 : BOOL ;
    E0998 : BOOL ;	//=CH2_4++ZNE05+TQ_01;PRÉ-ALARME DE CORREIA LENTA DE POSIÇÃO ALTA +TQ_01;58
    E0999 : BOOL ;	//=CH2_4++ZNE05+TQ_01;PRÉ-ALARME DA CORREIA LENTA POSIÇÃO BAIXA +TQ_01;58
    E1000 : BOOL ;
    E1001 : BOOL ;	//=CH2_4++ZNE05+TQ_01;PRÉ-ALARME DE BYPASS DE FALHA ATIVO;58
    E1002 : BOOL ;
    E1003 : BOOL ;
    E1004 : BOOL ;
    E1005 : BOOL ;
    E1006 : BOOL ;
    E1007 : BOOL ;
    E1008 : BOOL ;
    E1009 : BOOL ;
    E1010 : BOOL ;
    E1011 : BOOL ;
    E1012 : BOOL ;
    E1013 : BOOL ;
    E1014 : BOOL ;
    E1015 : BOOL ;
    E1016 : BOOL ;
    E1017 : BOOL ;	//=CH2_4++ZNE05+TQ_01;CICLO AUTOMÁTICO PASSO A PASSO INICIADO;58
    E1018 : BOOL ;
    E1019 : BOOL ;
    E1020 : BOOL ;
    E1021 : BOOL ;
    E1022 : BOOL ;
    E1023 : BOOL ;
    E1024 : BOOL ;
   END_STRUCT ;
  END_STRUCT ;
BEGIN
   CM_ID := '=CH1_2';
   STATION_ID := '++ZNE05';
   ELEMENT_ID := '';
   DB_ID := 0;
   PART_IDENTIFICATION := '';
   ACT_CYCLE_TIME := 0;
   COUNT_GOOD := 0;
   COUNT_SCRAP := 0;
   ACCUMULATORS[0] := 0;
   ACCUMULATORS[1] := 0;
   ACCUMULATORS[2] := 0;
   ACCUMULATORS[3] := 0;
   ACCUMULATORS[4] := 0;
   ACCUMULATORS[5] := 0;
   ACCUMULATORS[6] := 0;
   ACCUMULATORS[7] := 0;
   ACCUMULATORS[8] := 0;
   ACCUMULATORS[9] := 0;
   ACCUMULATORS[10] := 0;
   ACCUMULATORS[11] := 0;
   ACCUMULATORS[12] := 0;
   ACCUMULATORS[13] := 0;
   ACCUMULATORS[14] := 0;
   ACCUMULATORS[15] := 0;
   SPARE_01[0] := 0;
   SPARE_01[1] := 0;
   SPARE_01[2] := 0;
   SPARE_01[3] := 0;
   SPARE_01[4] := 0;
   SPARE_01[5] := 0;
   SPARE_01[6] := 0;
   SPARE_01[7] := 0;
   SPARE_01[8] := 0;
   SPARE_01[9] := 0;
   SPARE_01[10] := 0;
   SPARE_01[11] := 0;
   SPARE_01[12] := 0;
   SPARE_01[13] := 0;
   SPARE_01[14] := 0;
   SPARE_01[15] := 0;
   SPARE_01[16] := 0;
   SPARE_01[17] := 0;
   CODE_EVENT[0] := 0;
   CODE_EVENT[1] := 0;
   CODE_EVENT[2] := 0;
   CODE_EVENT[3] := 0;
   CODE_EVENT[4] := 0;
   CODE_EVENT[5] := 0;
   CODE_EVENT[6] := 0;
   CODE_EVENT[7] := 0;
   EVENTS.E0001 := FALSE;
   EVENTS.E0002 := FALSE;
   EVENTS.E0003 := FALSE;
   EVENTS.E0004 := FALSE;
   EVENTS.E0005 := FALSE;
   EVENTS.E0006 := FALSE;
   EVENTS.E0007 := FALSE;
   EVENTS.E0008 := FALSE;
   EVENTS.E0009 := FALSE;
   EVENTS.E0010 := FALSE;
   EVENTS.E0011 := FALSE;
   EVENTS.E0012 := FALSE;
   EVENTS.E0013 := FALSE;
   EVENTS.E0014 := FALSE;
   EVENTS.E0015 := FALSE;
   EVENTS.E0016 := FALSE;
   EVENTS.E0017 := FALSE;
   EVENTS.E0018 := FALSE;
   EVENTS.E0019 := FALSE;
   EVENTS.E0020 := FALSE;
   EVENTS.E0021 := FALSE;
   EVENTS.E0022 := FALSE;
   EVENTS.E0023 := FALSE;
   EVENTS.E0024 := FALSE;
   EVENTS.E0025 := FALSE;
   EVENTS.E0026 := FALSE;
   EVENTS.E0027 := FALSE;
   EVENTS.E0028 := FALSE;
   EVENTS.E0029 := FALSE;
   EVENTS.E0030 := FALSE;
   EVENTS.E0031 := FALSE;
   EVENTS.E0032 := FALSE;
   EVENTS.E0033 := FALSE;
   EVENTS.E0034 := FALSE;
   EVENTS.E0035 := FALSE;
   EVENTS.E0036 := FALSE;
   EVENTS.E0037 := FALSE;
   EVENTS.E0038 := FALSE;
   EVENTS.E0039 := FALSE;
   EVENTS.E0040 := FALSE;
   EVENTS.E0041 := FALSE;
   EVENTS.E0042 := FALSE;
   EVENTS.E0043 := FALSE;
   EVENTS.E0044 := FALSE;
   EVENTS.E0045 := FALSE;
   EVENTS.E0046 := FALSE;
   EVENTS.E0047 := FALSE;
   EVENTS.E0048 := FALSE;
   EVENTS.E0049 := FALSE;
   EVENTS.E0050 := FALSE;
   EVENTS.E0051 := FALSE;
   EVENTS.E0052 := FALSE;
   EVENTS.E0053 := FALSE;
   EVENTS.E0054 := FALSE;
   EVENTS.E0055 := FALSE;
   EVENTS.E0056 := FALSE;
   EVENTS.E0057 := FALSE;
   EVENTS.E0058 := FALSE;
   EVENTS.E0059 := FALSE;
   EVENTS.E0060 := FALSE;
   EVENTS.E0061 := FALSE;
   EVENTS.E0062 := FALSE;
   EVENTS.E0063 := FALSE;
   EVENTS.E0064 := FALSE;
   EVENTS.E0065 := FALSE;
   EVENTS.E0066 := FALSE;
   EVENTS.E0067 := FALSE;
   EVENTS.E0068 := FALSE;
   EVENTS.E0069 := FALSE;
   EVENTS.E0070 := FALSE;
   EVENTS.E0071 := FALSE;
   EVENTS.E0072 := FALSE;
   EVENTS.E0073 := FALSE;
   EVENTS.E0074 := FALSE;
   EVENTS.E0075 := FALSE;
   EVENTS.E0076 := FALSE;
   EVENTS.E0077 := FALSE;
   EVENTS.E0078 := FALSE;
   EVENTS.E0079 := FALSE;
   EVENTS.E0080 := FALSE;
   EVENTS.E0081 := FALSE;
   EVENTS.E0082 := FALSE;
   EVENTS.E0083 := FALSE;
   EVENTS.E0084 := FALSE;
   EVENTS.E0085 := FALSE;
   EVENTS.E0086 := FALSE;
   EVENTS.E0087 := FALSE;
   EVENTS.E0088 := FALSE;
   EVENTS.E0089 := FALSE;
   EVENTS.E0090 := FALSE;
   EVENTS.E0091 := FALSE;
   EVENTS.E0092 := FALSE;
   EVENTS.E0093 := FALSE;
   EVENTS.E0094 := FALSE;
   EVENTS.E0095 := FALSE;
   EVENTS.E0096 := FALSE;
   EVENTS.E0097 := FALSE;
   EVENTS.E0098 := FALSE;
   EVENTS.E0099 := FALSE;
   EVENTS.E0100 := FALSE;
   EVENTS.E0101 := FALSE;
   EVENTS.E0102 := FALSE;
   EVENTS.E0103 := FALSE;
   EVENTS.E0104 := FALSE;
   EVENTS.E0105 := FALSE;
   EVENTS.E0106 := FALSE;
   EVENTS.E0107 := FALSE;
   EVENTS.E0108 := FALSE;
   EVENTS.E0109 := FALSE;
   EVENTS.E0110 := FALSE;
   EVENTS.E0111 := FALSE;
   EVENTS.E0112 := FALSE;
   EVENTS.E0113 := FALSE;
   EVENTS.E0114 := FALSE;
   EVENTS.E0115 := FALSE;
   EVENTS.E0116 := FALSE;
   EVENTS.E0117 := FALSE;
   EVENTS.E0118 := FALSE;
   EVENTS.E0119 := FALSE;
   EVENTS.E0120 := FALSE;
   EVENTS.E0121 := FALSE;
   EVENTS.E0122 := FALSE;
   EVENTS.E0123 := FALSE;
   EVENTS.E0124 := FALSE;
   EVENTS.E0125 := FALSE;
   EVENTS.E0126 := FALSE;
   EVENTS.E0127 := FALSE;
   EVENTS.E0128 := FALSE;
   EVENTS.E0129 := FALSE;
   EVENTS.E0130 := FALSE;
   EVENTS.E0131 := FALSE;
   EVENTS.E0132 := FALSE;
   EVENTS.E0133 := FALSE;
   EVENTS.E0134 := FALSE;
   EVENTS.E0135 := FALSE;
   EVENTS.E0136 := FALSE;
   EVENTS.E0137 := FALSE;
   EVENTS.E0138 := FALSE;
   EVENTS.E0139 := FALSE;
   EVENTS.E0140 := FALSE;
   EVENTS.E0141 := FALSE;
   EVENTS.E0142 := FALSE;
   EVENTS.E0143 := FALSE;
   EVENTS.E0144 := FALSE;
   EVENTS.E0145 := FALSE;
   EVENTS.E0146 := FALSE;
   EVENTS.E0147 := FALSE;
   EVENTS.E0148 := FALSE;
   EVENTS.E0149 := FALSE;
   EVENTS.E0150 := FALSE;
   EVENTS.E0151 := FALSE;
   EVENTS.E0152 := FALSE;
   EVENTS.E0153 := FALSE;
   EVENTS.E0154 := FALSE;
   EVENTS.E0155 := FALSE;
   EVENTS.E0156 := FALSE;
   EVENTS.E0157 := FALSE;
   EVENTS.E0158 := FALSE;
   EVENTS.E0159 := FALSE;
   EVENTS.E0160 := FALSE;
   EVENTS.E0161 := FALSE;
   EVENTS.E0162 := FALSE;
   EVENTS.E0163 := FALSE;
   EVENTS.E0164 := FALSE;
   EVENTS.E0165 := FALSE;
   EVENTS.E0166 := FALSE;
   EVENTS.E0167 := FALSE;
   EVENTS.E0168 := FALSE;
   EVENTS.E0169 := FALSE;
   EVENTS.E0170 := FALSE;
   EVENTS.E0171 := FALSE;
   EVENTS.E0172 := FALSE;
   EVENTS.E0173 := FALSE;
   EVENTS.E0174 := FALSE;
   EVENTS.E0175 := FALSE;
   EVENTS.E0176 := FALSE;
   EVENTS.E0177 := FALSE;
   EVENTS.E0178 := FALSE;
   EVENTS.E0179 := FALSE;
   EVENTS.E0180 := FALSE;
   EVENTS.E0181 := FALSE;
   EVENTS.E0182 := FALSE;
   EVENTS.E0183 := FALSE;
   EVENTS.E0184 := FALSE;
   EVENTS.E0185 := FALSE;
   EVENTS.E0186 := FALSE;
   EVENTS.E0187 := FALSE;
   EVENTS.E0188 := FALSE;
   EVENTS.E0189 := FALSE;
   EVENTS.E0190 := FALSE;
   EVENTS.E0191 := FALSE;
   EVENTS.E0192 := FALSE;
   EVENTS.E0193 := FALSE;
   EVENTS.E0194 := FALSE;
   EVENTS.E0195 := FALSE;
   EVENTS.E0196 := FALSE;
   EVENTS.E0197 := FALSE;
   EVENTS.E0198 := FALSE;
   EVENTS.E0199 := FALSE;
   EVENTS.E0200 := FALSE;
   EVENTS.E0201 := FALSE;
   EVENTS.E0202 := FALSE;
   EVENTS.E0203 := FALSE;
   EVENTS.E0204 := FALSE;
   EVENTS.E0205 := FALSE;
   EVENTS.E0206 := FALSE;
   EVENTS.E0207 := FALSE;
   EVENTS.E0208 := FALSE;
   EVENTS.E0209 := FALSE;
   EVENTS.E0210 := FALSE;
   EVENTS.E0211 := FALSE;
   EVENTS.E0212 := FALSE;
   EVENTS.E0213 := FALSE;
   EVENTS.E0214 := FALSE;
   EVENTS.E0215 := FALSE;
   EVENTS.E0216 := FALSE;
   EVENTS.E0217 := FALSE;
   EVENTS.E0218 := FALSE;
   EVENTS.E0219 := FALSE;
   EVENTS.E0220 := FALSE;
   EVENTS.E0221 := FALSE;
   EVENTS.E0222 := FALSE;
   EVENTS.E0223 := FALSE;
   EVENTS.E0224 := FALSE;
   EVENTS.E0225 := FALSE;
   EVENTS.E0226 := FALSE;
   EVENTS.E0227 := FALSE;
   EVENTS.E0228 := FALSE;
   EVENTS.E0229 := FALSE;
   EVENTS.E0230 := FALSE;
   EVENTS.E0231 := FALSE;
   EVENTS.E0232 := FALSE;
   EVENTS.E0233 := FALSE;
   EVENTS.E0234 := FALSE;
   EVENTS.E0235 := FALSE;
   EVENTS.E0236 := FALSE;
   EVENTS.E0237 := FALSE;
   EVENTS.E0238 := FALSE;
   EVENTS.E0239 := FALSE;
   EVENTS.E0240 := FALSE;
   EVENTS.E0241 := FALSE;
   EVENTS.E0242 := FALSE;
   EVENTS.E0243 := FALSE;
   EVENTS.E0244 := FALSE;
   EVENTS.E0245 := FALSE;
   EVENTS.E0246 := FALSE;
   EVENTS.E0247 := FALSE;
   EVENTS.E0248 := FALSE;
   EVENTS.E0249 := FALSE;
   EVENTS.E0250 := FALSE;
   EVENTS.E0251 := FALSE;
   EVENTS.E0252 := FALSE;
   EVENTS.E0253 := FALSE;
   EVENTS.E0254 := FALSE;
   EVENTS.E0255 := FALSE;
   EVENTS.E0256 := FALSE;
   EVENTS.E0257 := FALSE;
   EVENTS.E0258 := FALSE;
   EVENTS.E0259 := FALSE;
   EVENTS.E0260 := FALSE;
   EVENTS.E0261 := FALSE;
   EVENTS.E0262 := FALSE;
   EVENTS.E0263 := FALSE;
   EVENTS.E0264 := FALSE;
   EVENTS.E0265 := FALSE;
   EVENTS.E0266 := FALSE;
   EVENTS.E0267 := FALSE;
   EVENTS.E0268 := FALSE;
   EVENTS.E0269 := FALSE;
   EVENTS.E0270 := FALSE;
   EVENTS.E0271 := FALSE;
   EVENTS.E0272 := FALSE;
   EVENTS.E0273 := FALSE;
   EVENTS.E0274 := FALSE;
   EVENTS.E0275 := FALSE;
   EVENTS.E0276 := FALSE;
   EVENTS.E0277 := FALSE;
   EVENTS.E0278 := FALSE;
   EVENTS.E0279 := FALSE;
   EVENTS.E0280 := FALSE;
   EVENTS.E0281 := FALSE;
   EVENTS.E0282 := FALSE;
   EVENTS.E0283 := FALSE;
   EVENTS.E0284 := FALSE;
   EVENTS.E0285 := FALSE;
   EVENTS.E0286 := FALSE;
   EVENTS.E0287 := FALSE;
   EVENTS.E0288 := FALSE;
   EVENTS.E0289 := FALSE;
   EVENTS.E0290 := FALSE;
   EVENTS.E0291 := FALSE;
   EVENTS.E0292 := FALSE;
   EVENTS.E0293 := FALSE;
   EVENTS.E0294 := FALSE;
   EVENTS.E0295 := FALSE;
   EVENTS.E0296 := FALSE;
   EVENTS.E0297 := FALSE;
   EVENTS.E0298 := FALSE;
   EVENTS.E0299 := FALSE;
   EVENTS.E0300 := FALSE;
   EVENTS.E0301 := FALSE;
   EVENTS.E0302 := FALSE;
   EVENTS.E0303 := FALSE;
   EVENTS.E0304 := FALSE;
   EVENTS.E0305 := TRUE;
   EVENTS.E0306 := FALSE;
   EVENTS.E0307 := FALSE;
   EVENTS.E0308 := FALSE;
   EVENTS.E0309 := FALSE;
   EVENTS.E0310 := FALSE;
   EVENTS.E0311 := FALSE;
   EVENTS.E0312 := FALSE;
   EVENTS.E0313 := FALSE;
   EVENTS.E0314 := FALSE;
   EVENTS.E0315 := FALSE;
   EVENTS.E0316 := FALSE;
   EVENTS.E0317 := FALSE;
   EVENTS.E0318 := FALSE;
   EVENTS.E0319 := FALSE;
   EVENTS.E0320 := FALSE;
   EVENTS.E0321 := FALSE;
   EVENTS.E0322 := FALSE;
   EVENTS.E0323 := FALSE;
   EVENTS.E0324 := FALSE;
   EVENTS.E0325 := FALSE;
   EVENTS.E0326 := FALSE;
   EVENTS.E0327 := FALSE;
   EVENTS.E0328 := FALSE;
   EVENTS.E0329 := FALSE;
   EVENTS.E0330 := FALSE;
   EVENTS.E0331 := FALSE;
   EVENTS.E0332 := FALSE;
   EVENTS.E0333 := FALSE;
   EVENTS.E0334 := FALSE;
   EVENTS.E0335 := FALSE;
   EVENTS.E0336 := FALSE;
   EVENTS.E0337 := FALSE;
   EVENTS.E0338 := FALSE;
   EVENTS.E0339 := FALSE;
   EVENTS.E0340 := FALSE;
   EVENTS.E0341 := FALSE;
   EVENTS.E0342 := FALSE;
   EVENTS.E0343 := FALSE;
   EVENTS.E0344 := FALSE;
   EVENTS.E0345 := FALSE;
   EVENTS.E0346 := FALSE;
   EVENTS.E0347 := FALSE;
   EVENTS.E0348 := FALSE;
   EVENTS.E0349 := FALSE;
   EVENTS.E0350 := FALSE;
   EVENTS.E0351 := FALSE;
   EVENTS.E0352 := FALSE;
   EVENTS.E0353 := FALSE;
   EVENTS.E0354 := FALSE;
   EVENTS.E0355 := FALSE;
   EVENTS.E0356 := FALSE;
   EVENTS.E0357 := FALSE;
   EVENTS.E0358 := FALSE;
   EVENTS.E0359 := FALSE;
   EVENTS.E0360 := FALSE;
   EVENTS.E0361 := FALSE;
   EVENTS.E0362 := FALSE;
   EVENTS.E0363 := FALSE;
   EVENTS.E0364 := FALSE;
   EVENTS.E0365 := FALSE;
   EVENTS.E0366 := FALSE;
   EVENTS.E0367 := FALSE;
   EVENTS.E0368 := FALSE;
   EVENTS.E0369 := FALSE;
   EVENTS.E0370 := FALSE;
   EVENTS.E0371 := FALSE;
   EVENTS.E0372 := FALSE;
   EVENTS.E0373 := FALSE;
   EVENTS.E0374 := FALSE;
   EVENTS.E0375 := FALSE;
   EVENTS.E0376 := FALSE;
   EVENTS.E0377 := FALSE;
   EVENTS.E0378 := FALSE;
   EVENTS.E0379 := FALSE;
   EVENTS.E0380 := FALSE;
   EVENTS.E0381 := FALSE;
   EVENTS.E0382 := FALSE;
   EVENTS.E0383 := FALSE;
   EVENTS.E0384 := FALSE;
   EVENTS.E0385 := FALSE;
   EVENTS.E0386 := FALSE;
   EVENTS.E0387 := FALSE;
   EVENTS.E0388 := FALSE;
   EVENTS.E0389 := FALSE;
   EVENTS.E0390 := FALSE;
   EVENTS.E0391 := FALSE;
   EVENTS.E0392 := FALSE;
   EVENTS.E0393 := FALSE;
   EVENTS.E0394 := FALSE;
   EVENTS.E0395 := FALSE;
   EVENTS.E0396 := FALSE;
   EVENTS.E0397 := FALSE;
   EVENTS.E0398 := FALSE;
   EVENTS.E0399 := FALSE;
   EVENTS.E0400 := FALSE;
   EVENTS.E0401 := FALSE;
   EVENTS.E0402 := FALSE;
   EVENTS.E0403 := FALSE;
   EVENTS.E0404 := FALSE;
   EVENTS.E0405 := FALSE;
   EVENTS.E0406 := FALSE;
   EVENTS.E0407 := FALSE;
   EVENTS.E0408 := FALSE;
   EVENTS.E0409 := FALSE;
   EVENTS.E0410 := FALSE;
   EVENTS.E0411 := FALSE;
   EVENTS.E0412 := FALSE;
   EVENTS.E0413 := FALSE;
   EVENTS.E0414 := FALSE;
   EVENTS.E0415 := FALSE;
   EVENTS.E0416 := FALSE;
   EVENTS.E0417 := FALSE;
   EVENTS.E0418 := FALSE;
   EVENTS.E0419 := FALSE;
   EVENTS.E0420 := FALSE;
   EVENTS.E0421 := FALSE;
   EVENTS.E0422 := FALSE;
   EVENTS.E0423 := FALSE;
   EVENTS.E0424 := FALSE;
   EVENTS.E0425 := FALSE;
   EVENTS.E0426 := FALSE;
   EVENTS.E0427 := FALSE;
   EVENTS.E0428 := FALSE;
   EVENTS.E0429 := FALSE;
   EVENTS.E0430 := FALSE;
   EVENTS.E0431 := FALSE;
   EVENTS.E0432 := FALSE;
   EVENTS.E0433 := FALSE;
   EVENTS.E0434 := FALSE;
   EVENTS.E0435 := FALSE;
   EVENTS.E0436 := FALSE;
   EVENTS.E0437 := FALSE;
   EVENTS.E0438 := FALSE;
   EVENTS.E0439 := FALSE;
   EVENTS.E0440 := FALSE;
   EVENTS.E0441 := FALSE;
   EVENTS.E0442 := FALSE;
   EVENTS.E0443 := FALSE;
   EVENTS.E0444 := FALSE;
   EVENTS.E0445 := FALSE;
   EVENTS.E0446 := FALSE;
   EVENTS.E0447 := FALSE;
   EVENTS.E0448 := FALSE;
   EVENTS.E0449 := FALSE;
   EVENTS.E0450 := FALSE;
   EVENTS.E0451 := FALSE;
   EVENTS.E0452 := FALSE;
   EVENTS.E0453 := FALSE;
   EVENTS.E0454 := FALSE;
   EVENTS.E0455 := FALSE;
   EVENTS.E0456 := FALSE;
   EVENTS.E0457 := FALSE;
   EVENTS.E0458 := FALSE;
   EVENTS.E0459 := FALSE;
   EVENTS.E0460 := FALSE;
   EVENTS.E0461 := FALSE;
   EVENTS.E0462 := FALSE;
   EVENTS.E0463 := FALSE;
   EVENTS.E0464 := FALSE;
   EVENTS.E0465 := FALSE;
   EVENTS.E0466 := FALSE;
   EVENTS.E0467 := FALSE;
   EVENTS.E0468 := FALSE;
   EVENTS.E0469 := FALSE;
   EVENTS.E0470 := FALSE;
   EVENTS.E0471 := FALSE;
   EVENTS.E0472 := FALSE;
   EVENTS.E0473 := FALSE;
   EVENTS.E0474 := FALSE;
   EVENTS.E0475 := FALSE;
   EVENTS.E0476 := FALSE;
   EVENTS.E0477 := FALSE;
   EVENTS.E0478 := FALSE;
   EVENTS.E0479 := FALSE;
   EVENTS.E0480 := FALSE;
   EVENTS.E0481 := FALSE;
   EVENTS.E0482 := FALSE;
   EVENTS.E0483 := FALSE;
   EVENTS.E0484 := FALSE;
   EVENTS.E0485 := FALSE;
   EVENTS.E0486 := FALSE;
   EVENTS.E0487 := FALSE;
   EVENTS.E0488 := FALSE;
   EVENTS.E0489 := FALSE;
   EVENTS.E0490 := FALSE;
   EVENTS.E0491 := FALSE;
   EVENTS.E0492 := FALSE;
   EVENTS.E0493 := FALSE;
   EVENTS.E0494 := FALSE;
   EVENTS.E0495 := FALSE;
   EVENTS.E0496 := FALSE;
   EVENTS.E0497 := FALSE;
   EVENTS.E0498 := FALSE;
   EVENTS.E0499 := FALSE;
   EVENTS.E0500 := FALSE;
   EVENTS.E0501 := FALSE;
   EVENTS.E0502 := FALSE;
   EVENTS.E0503 := FALSE;
   EVENTS.E0504 := FALSE;
   EVENTS.E0505 := FALSE;
   EVENTS.E0506 := FALSE;
   EVENTS.E0507 := FALSE;
   EVENTS.E0508 := FALSE;
   EVENTS.E0509 := FALSE;
   EVENTS.E0510 := FALSE;
   EVENTS.E0511 := FALSE;
   EVENTS.E0512 := FALSE;
   EVENTS.E0513 := FALSE;
   EVENTS.E0514 := FALSE;
   EVENTS.E0515 := FALSE;
   EVENTS.E0516 := FALSE;
   EVENTS.E0517 := FALSE;
   EVENTS.E0518 := FALSE;
   EVENTS.E0519 := FALSE;
   EVENTS.E0520 := FALSE;
   EVENTS.E0521 := FALSE;
   EVENTS.E0522 := FALSE;
   EVENTS.E0523 := FALSE;
   EVENTS.E0524 := FALSE;
   EVENTS.E0525 := FALSE;
   EVENTS.E0526 := FALSE;
   EVENTS.E0527 := FALSE;
   EVENTS.E0528 := FALSE;
   EVENTS.E0529 := FALSE;
   EVENTS.E0530 := FALSE;
   EVENTS.E0531 := FALSE;
   EVENTS.E0532 := FALSE;
   EVENTS.E0533 := FALSE;
   EVENTS.E0534 := FALSE;
   EVENTS.E0535 := FALSE;
   EVENTS.E0536 := FALSE;
   EVENTS.E0537 := FALSE;
   EVENTS.E0538 := FALSE;
   EVENTS.E0539 := FALSE;
   EVENTS.E0540 := FALSE;
   EVENTS.E0541 := FALSE;
   EVENTS.E0542 := FALSE;
   EVENTS.E0543 := FALSE;
   EVENTS.E0544 := FALSE;
   EVENTS.E0545 := FALSE;
   EVENTS.E0546 := FALSE;
   EVENTS.E0547 := FALSE;
   EVENTS.E0548 := FALSE;
   EVENTS.E0549 := FALSE;
   EVENTS.E0550 := FALSE;
   EVENTS.E0551 := FALSE;
   EVENTS.E0552 := FALSE;
   EVENTS.E0553 := FALSE;
   EVENTS.E0554 := FALSE;
   EVENTS.E0555 := FALSE;
   EVENTS.E0556 := FALSE;
   EVENTS.E0557 := FALSE;
   EVENTS.E0558 := FALSE;
   EVENTS.E0559 := FALSE;
   EVENTS.E0560 := FALSE;
   EVENTS.E0561 := FALSE;
   EVENTS.E0562 := FALSE;
   EVENTS.E0563 := FALSE;
   EVENTS.E0564 := FALSE;
   EVENTS.E0565 := FALSE;
   EVENTS.E0566 := FALSE;
   EVENTS.E0567 := FALSE;
   EVENTS.E0568 := FALSE;
   EVENTS.E0569 := FALSE;
   EVENTS.E0570 := FALSE;
   EVENTS.E0571 := FALSE;
   EVENTS.E0572 := FALSE;
   EVENTS.E0573 := FALSE;
   EVENTS.E0574 := FALSE;
   EVENTS.E0575 := FALSE;
   EVENTS.E0576 := FALSE;
   EVENTS.E0577 := FALSE;
   EVENTS.E0578 := FALSE;
   EVENTS.E0579 := FALSE;
   EVENTS.E0580 := FALSE;
   EVENTS.E0581 := FALSE;
   EVENTS.E0582 := FALSE;
   EVENTS.E0583 := FALSE;
   EVENTS.E0584 := FALSE;
   EVENTS.E0585 := FALSE;
   EVENTS.E0586 := FALSE;
   EVENTS.E0587 := FALSE;
   EVENTS.E0588 := FALSE;
   EVENTS.E0589 := FALSE;
   EVENTS.E0590 := FALSE;
   EVENTS.E0591 := FALSE;
   EVENTS.E0592 := FALSE;
   EVENTS.E0593 := FALSE;
   EVENTS.E0594 := FALSE;
   EVENTS.E0595 := FALSE;
   EVENTS.E0596 := FALSE;
   EVENTS.E0597 := FALSE;
   EVENTS.E0598 := FALSE;
   EVENTS.E0599 := FALSE;
   EVENTS.E0600 := FALSE;
   EVENTS.E0601 := FALSE;
   EVENTS.E0602 := FALSE;
   EVENTS.E0603 := FALSE;
   EVENTS.E0604 := FALSE;
   EVENTS.E0605 := FALSE;
   EVENTS.E0606 := FALSE;
   EVENTS.E0607 := FALSE;
   EVENTS.E0608 := FALSE;
   EVENTS.E0609 := FALSE;
   EVENTS.E0610 := FALSE;
   EVENTS.E0611 := FALSE;
   EVENTS.E0612 := FALSE;
   EVENTS.E0613 := FALSE;
   EVENTS.E0614 := FALSE;
   EVENTS.E0615 := FALSE;
   EVENTS.E0616 := FALSE;
   EVENTS.E0617 := FALSE;
   EVENTS.E0618 := FALSE;
   EVENTS.E0619 := FALSE;
   EVENTS.E0620 := FALSE;
   EVENTS.E0621 := FALSE;
   EVENTS.E0622 := FALSE;
   EVENTS.E0623 := FALSE;
   EVENTS.E0624 := FALSE;
   EVENTS.E0625 := FALSE;
   EVENTS.E0626 := FALSE;
   EVENTS.E0627 := FALSE;
   EVENTS.E0628 := FALSE;
   EVENTS.E0629 := FALSE;
   EVENTS.E0630 := FALSE;
   EVENTS.E0631 := FALSE;
   EVENTS.E0632 := FALSE;
   EVENTS.E0633 := FALSE;
   EVENTS.E0634 := FALSE;
   EVENTS.E0635 := FALSE;
   EVENTS.E0636 := FALSE;
   EVENTS.E0637 := FALSE;
   EVENTS.E0638 := FALSE;
   EVENTS.E0639 := FALSE;
   EVENTS.E0640 := FALSE;
   EVENTS.E0641 := FALSE;
   EVENTS.E0642 := FALSE;
   EVENTS.E0643 := FALSE;
   EVENTS.E0644 := FALSE;
   EVENTS.E0645 := FALSE;
   EVENTS.E0646 := FALSE;
   EVENTS.E0647 := FALSE;
   EVENTS.E0648 := FALSE;
   EVENTS.E0649 := FALSE;
   EVENTS.E0650 := FALSE;
   EVENTS.E0651 := FALSE;
   EVENTS.E0652 := FALSE;
   EVENTS.E0653 := FALSE;
   EVENTS.E0654 := FALSE;
   EVENTS.E0655 := FALSE;
   EVENTS.E0656 := FALSE;
   EVENTS.E0657 := FALSE;
   EVENTS.E0658 := FALSE;
   EVENTS.E0659 := FALSE;
   EVENTS.E0660 := FALSE;
   EVENTS.E0661 := FALSE;
   EVENTS.E0662 := FALSE;
   EVENTS.E0663 := FALSE;
   EVENTS.E0664 := FALSE;
   EVENTS.E0665 := FALSE;
   EVENTS.E0666 := FALSE;
   EVENTS.E0667 := FALSE;
   EVENTS.E0668 := FALSE;
   EVENTS.E0669 := FALSE;
   EVENTS.E0670 := FALSE;
   EVENTS.E0671 := FALSE;
   EVENTS.E0672 := FALSE;
   EVENTS.E0673 := FALSE;
   EVENTS.E0674 := FALSE;
   EVENTS.E0675 := FALSE;
   EVENTS.E0676 := FALSE;
   EVENTS.E0677 := FALSE;
   EVENTS.E0678 := FALSE;
   EVENTS.E0679 := FALSE;
   EVENTS.E0680 := FALSE;
   EVENTS.E0681 := FALSE;
   EVENTS.E0682 := FALSE;
   EVENTS.E0683 := FALSE;
   EVENTS.E0684 := FALSE;
   EVENTS.E0685 := FALSE;
   EVENTS.E0686 := FALSE;
   EVENTS.E0687 := FALSE;
   EVENTS.E0688 := FALSE;
   EVENTS.E0689 := FALSE;
   EVENTS.E0690 := FALSE;
   EVENTS.E0691 := FALSE;
   EVENTS.E0692 := FALSE;
   EVENTS.E0693 := FALSE;
   EVENTS.E0694 := FALSE;
   EVENTS.E0695 := FALSE;
   EVENTS.E0696 := FALSE;
   EVENTS.E0697 := FALSE;
   EVENTS.E0698 := FALSE;
   EVENTS.E0699 := FALSE;
   EVENTS.E0700 := FALSE;
   EVENTS.E0701 := FALSE;
   EVENTS.E0702 := FALSE;
   EVENTS.E0703 := FALSE;
   EVENTS.E0704 := FALSE;
   EVENTS.E0705 := FALSE;
   EVENTS.E0706 := FALSE;
   EVENTS.E0707 := FALSE;
   EVENTS.E0708 := FALSE;
   EVENTS.E0709 := FALSE;
   EVENTS.E0710 := FALSE;
   EVENTS.E0711 := FALSE;
   EVENTS.E0712 := FALSE;
   EVENTS.E0713 := FALSE;
   EVENTS.E0714 := FALSE;
   EVENTS.E0715 := FALSE;
   EVENTS.E0716 := FALSE;
   EVENTS.E0717 := FALSE;
   EVENTS.E0718 := FALSE;
   EVENTS.E0719 := FALSE;
   EVENTS.E0720 := FALSE;
   EVENTS.E0721 := FALSE;
   EVENTS.E0722 := FALSE;
   EVENTS.E0723 := FALSE;
   EVENTS.E0724 := FALSE;
   EVENTS.E0725 := FALSE;
   EVENTS.E0726 := FALSE;
   EVENTS.E0727 := FALSE;
   EVENTS.E0728 := FALSE;
   EVENTS.E0729 := FALSE;
   EVENTS.E0730 := FALSE;
   EVENTS.E0731 := FALSE;
   EVENTS.E0732 := FALSE;
   EVENTS.E0733 := FALSE;
   EVENTS.E0734 := FALSE;
   EVENTS.E0735 := FALSE;
   EVENTS.E0736 := FALSE;
   EVENTS.E0737 := FALSE;
   EVENTS.E0738 := FALSE;
   EVENTS.E0739 := FALSE;
   EVENTS.E0740 := FALSE;
   EVENTS.E0741 := FALSE;
   EVENTS.E0742 := FALSE;
   EVENTS.E0743 := FALSE;
   EVENTS.E0744 := FALSE;
   EVENTS.E0745 := FALSE;
   EVENTS.E0746 := FALSE;
   EVENTS.E0747 := FALSE;
   EVENTS.E0748 := FALSE;
   EVENTS.E0749 := FALSE;
   EVENTS.E0750 := FALSE;
   EVENTS.E0751 := FALSE;
   EVENTS.E0752 := FALSE;
   EVENTS.E0753 := FALSE;
   EVENTS.E0754 := FALSE;
   EVENTS.E0755 := FALSE;
   EVENTS.E0756 := FALSE;
   EVENTS.E0757 := FALSE;
   EVENTS.E0758 := FALSE;
   EVENTS.E0759 := FALSE;
   EVENTS.E0760 := FALSE;
   EVENTS.E0761 := FALSE;
   EVENTS.E0762 := FALSE;
   EVENTS.E0763 := FALSE;
   EVENTS.E0764 := FALSE;
   EVENTS.E0765 := FALSE;
   EVENTS.E0766 := FALSE;
   EVENTS.E0767 := FALSE;
   EVENTS.E0768 := FALSE;
   EVENTS.E0769 := FALSE;
   EVENTS.E0770 := FALSE;
   EVENTS.E0771 := FALSE;
   EVENTS.E0772 := FALSE;
   EVENTS.E0773 := FALSE;
   EVENTS.E0774 := FALSE;
   EVENTS.E0775 := FALSE;
   EVENTS.E0776 := FALSE;
   EVENTS.E0777 := FALSE;
   EVENTS.E0778 := FALSE;
   EVENTS.E0779 := FALSE;
   EVENTS.E0780 := FALSE;
   EVENTS.E0781 := FALSE;
   EVENTS.E0782 := FALSE;
   EVENTS.E0783 := FALSE;
   EVENTS.E0784 := FALSE;
   EVENTS.E0785 := FALSE;
   EVENTS.E0786 := FALSE;
   EVENTS.E0787 := FALSE;
   EVENTS.E0788 := FALSE;
   EVENTS.E0789 := FALSE;
   EVENTS.E0790 := FALSE;
   EVENTS.E0791 := FALSE;
   EVENTS.E0792 := FALSE;
   EVENTS.E0793 := FALSE;
   EVENTS.E0794 := FALSE;
   EVENTS.E0795 := FALSE;
   EVENTS.E0796 := FALSE;
   EVENTS.E0797 := FALSE;
   EVENTS.E0798 := FALSE;
   EVENTS.E0799 := FALSE;
   EVENTS.E0800 := FALSE;
   EVENTS.E0801 := FALSE;
   EVENTS.E0802 := FALSE;
   EVENTS.E0803 := FALSE;
   EVENTS.E0804 := FALSE;
   EVENTS.E0805 := FALSE;
   EVENTS.E0806 := FALSE;
   EVENTS.E0807 := FALSE;
   EVENTS.E0808 := FALSE;
   EVENTS.E0809 := FALSE;
   EVENTS.E0810 := FALSE;
   EVENTS.E0811 := FALSE;
   EVENTS.E0812 := FALSE;
   EVENTS.E0813 := FALSE;
   EVENTS.E0814 := FALSE;
   EVENTS.E0815 := FALSE;
   EVENTS.E0816 := FALSE;
   EVENTS.E0817 := FALSE;
   EVENTS.E0818 := FALSE;
   EVENTS.E0819 := FALSE;
   EVENTS.E0820 := FALSE;
   EVENTS.E0821 := FALSE;
   EVENTS.E0822 := FALSE;
   EVENTS.E0823 := FALSE;
   EVENTS.E0824 := FALSE;
   EVENTS.E0825 := FALSE;
   EVENTS.E0826 := FALSE;
   EVENTS.E0827 := FALSE;
   EVENTS.E0828 := FALSE;
   EVENTS.E0829 := FALSE;
   EVENTS.E0830 := FALSE;
   EVENTS.E0831 := FALSE;
   EVENTS.E0832 := FALSE;
   EVENTS.E0833 := FALSE;
   EVENTS.E0834 := FALSE;
   EVENTS.E0835 := FALSE;
   EVENTS.E0836 := FALSE;
   EVENTS.E0837 := FALSE;
   EVENTS.E0838 := FALSE;
   EVENTS.E0839 := FALSE;
   EVENTS.E0840 := FALSE;
   EVENTS.E0841 := FALSE;
   EVENTS.E0842 := FALSE;
   EVENTS.E0843 := FALSE;
   EVENTS.E0844 := FALSE;
   EVENTS.E0845 := FALSE;
   EVENTS.E0846 := FALSE;
   EVENTS.E0847 := FALSE;
   EVENTS.E0848 := FALSE;
   EVENTS.E0849 := FALSE;
   EVENTS.E0850 := FALSE;
   EVENTS.E0851 := FALSE;
   EVENTS.E0852 := FALSE;
   EVENTS.E0853 := FALSE;
   EVENTS.E0854 := FALSE;
   EVENTS.E0855 := FALSE;
   EVENTS.E0856 := FALSE;
   EVENTS.E0857 := FALSE;
   EVENTS.E0858 := FALSE;
   EVENTS.E0859 := FALSE;
   EVENTS.E0860 := FALSE;
   EVENTS.E0861 := FALSE;
   EVENTS.E0862 := FALSE;
   EVENTS.E0863 := FALSE;
   EVENTS.E0864 := FALSE;
   EVENTS.E0865 := FALSE;
   EVENTS.E0866 := FALSE;
   EVENTS.E0867 := FALSE;
   EVENTS.E0868 := FALSE;
   EVENTS.E0869 := FALSE;
   EVENTS.E0870 := FALSE;
   EVENTS.E0871 := FALSE;
   EVENTS.E0872 := FALSE;
   EVENTS.E0873 := FALSE;
   EVENTS.E0874 := FALSE;
   EVENTS.E0875 := FALSE;
   EVENTS.E0876 := FALSE;
   EVENTS.E0877 := FALSE;
   EVENTS.E0878 := FALSE;
   EVENTS.E0879 := FALSE;
   EVENTS.E0880 := FALSE;
   EVENTS.E0881 := FALSE;
   EVENTS.E0882 := FALSE;
   EVENTS.E0883 := FALSE;
   EVENTS.E0884 := FALSE;
   EVENTS.E0885 := FALSE;
   EVENTS.E0886 := FALSE;
   EVENTS.E0887 := FALSE;
   EVENTS.E0888 := FALSE;
   EVENTS.E0889 := FALSE;
   EVENTS.E0890 := FALSE;
   EVENTS.E0891 := FALSE;
   EVENTS.E0892 := FALSE;
   EVENTS.E0893 := FALSE;
   EVENTS.E0894 := FALSE;
   EVENTS.E0895 := FALSE;
   EVENTS.E0896 := FALSE;
   EVENTS.E0897 := FALSE;
   EVENTS.E0898 := FALSE;
   EVENTS.E0899 := FALSE;
   EVENTS.E0900 := FALSE;
   EVENTS.E0901 := FALSE;
   EVENTS.E0902 := FALSE;
   EVENTS.E0903 := FALSE;
   EVENTS.E0904 := FALSE;
   EVENTS.E0905 := FALSE;
   EVENTS.E0906 := FALSE;
   EVENTS.E0907 := FALSE;
   EVENTS.E0908 := FALSE;
   EVENTS.E0909 := FALSE;
   EVENTS.E0910 := FALSE;
   EVENTS.E0911 := FALSE;
   EVENTS.E0912 := FALSE;
   EVENTS.E0913 := FALSE;
   EVENTS.E0914 := FALSE;
   EVENTS.E0915 := FALSE;
   EVENTS.E0916 := FALSE;
   EVENTS.E0917 := FALSE;
   EVENTS.E0918 := FALSE;
   EVENTS.E0919 := FALSE;
   EVENTS.E0920 := FALSE;
   EVENTS.E0921 := FALSE;
   EVENTS.E0922 := FALSE;
   EVENTS.E0923 := FALSE;
   EVENTS.E0924 := FALSE;
   EVENTS.E0925 := FALSE;
   EVENTS.E0926 := FALSE;
   EVENTS.E0927 := FALSE;
   EVENTS.E0928 := FALSE;
   EVENTS.E0929 := FALSE;
   EVENTS.E0930 := FALSE;
   EVENTS.E0931 := FALSE;
   EVENTS.E0932 := FALSE;
   EVENTS.E0933 := FALSE;
   EVENTS.E0934 := FALSE;
   EVENTS.E0935 := FALSE;
   EVENTS.E0936 := FALSE;
   EVENTS.E0937 := FALSE;
   EVENTS.E0938 := FALSE;
   EVENTS.E0939 := FALSE;
   EVENTS.E0940 := FALSE;
   EVENTS.E0941 := FALSE;
   EVENTS.E0942 := FALSE;
   EVENTS.E0943 := FALSE;
   EVENTS.E0944 := FALSE;
   EVENTS.E0945 := FALSE;
   EVENTS.E0946 := FALSE;
   EVENTS.E0947 := FALSE;
   EVENTS.E0948 := FALSE;
   EVENTS.E0949 := FALSE;
   EVENTS.E0950 := FALSE;
   EVENTS.E0951 := FALSE;
   EVENTS.E0952 := FALSE;
   EVENTS.E0953 := FALSE;
   EVENTS.E0954 := FALSE;
   EVENTS.E0955 := FALSE;
   EVENTS.E0956 := FALSE;
   EVENTS.E0957 := FALSE;
   EVENTS.E0958 := FALSE;
   EVENTS.E0959 := FALSE;
   EVENTS.E0960 := FALSE;
   EVENTS.E0961 := FALSE;
   EVENTS.E0962 := FALSE;
   EVENTS.E0963 := FALSE;
   EVENTS.E0964 := FALSE;
   EVENTS.E0965 := FALSE;
   EVENTS.E0966 := FALSE;
   EVENTS.E0967 := FALSE;
   EVENTS.E0968 := FALSE;
   EVENTS.E0969 := FALSE;
   EVENTS.E0970 := FALSE;
   EVENTS.E0971 := FALSE;
   EVENTS.E0972 := FALSE;
   EVENTS.E0973 := FALSE;
   EVENTS.E0974 := FALSE;
   EVENTS.E0975 := FALSE;
   EVENTS.E0976 := FALSE;
   EVENTS.E0977 := FALSE;
   EVENTS.E0978 := FALSE;
   EVENTS.E0979 := FALSE;
   EVENTS.E0980 := FALSE;
   EVENTS.E0981 := FALSE;
   EVENTS.E0982 := FALSE;
   EVENTS.E0983 := FALSE;
   EVENTS.E0984 := FALSE;
   EVENTS.E0985 := FALSE;
   EVENTS.E0986 := FALSE;
   EVENTS.E0987 := FALSE;
   EVENTS.E0988 := FALSE;
   EVENTS.E0989 := FALSE;
   EVENTS.E0990 := FALSE;
   EVENTS.E0991 := FALSE;
   EVENTS.E0992 := FALSE;
   EVENTS.E0993 := FALSE;
   EVENTS.E0994 := FALSE;
   EVENTS.E0995 := FALSE;
   EVENTS.E0996 := FALSE;
   EVENTS.E0997 := FALSE;
   EVENTS.E0998 := TRUE;
   EVENTS.E0999 := FALSE;
   EVENTS.E1000 := FALSE;
   EVENTS.E1001 := FALSE;
   EVENTS.E1002 := FALSE;
   EVENTS.E1003 := FALSE;
   EVENTS.E1004 := FALSE;
   EVENTS.E1005 := FALSE;
   EVENTS.E1006 := FALSE;
   EVENTS.E1007 := FALSE;
   EVENTS.E1008 := FALSE;
   EVENTS.E1009 := FALSE;
   EVENTS.E1010 := FALSE;
   EVENTS.E1011 := FALSE;
   EVENTS.E1012 := FALSE;
   EVENTS.E1013 := FALSE;
   EVENTS.E1014 := FALSE;
   EVENTS.E1015 := FALSE;
   EVENTS.E1016 := FALSE;
   EVENTS.E1017 := FALSE;
   EVENTS.E1018 := FALSE;
   EVENTS.E1019 := FALSE;
   EVENTS.E1020 := FALSE;
   EVENTS.E1021 := FALSE;
   EVENTS.E1022 := FALSE;
   EVENTS.E1023 := FALSE;
   EVENTS.E1024 := FALSE;
END_DATA_BLOCK
